HMI tags "2930RS001A01L01"
   "2930RS001A01L01.MSW" : 52809b66-421d-457f-8884-6f7a49d4e247 AT %DB5093.DBX18.0, 500 ms
   "2930RS001A01L01.DefaultText" : TextRef, internal   // Заголовок POPUP окна. При експорте из ECS через скрипт заполняется автоматически, если теги копируются в ручную то требуется в ручную задатать свойство Start Value
   "2930RS001A01L01.BlockInfo" : Array [0..2] of Int AT %DB5093.DBX38.0, 500 ms
   "2930RS001A01L01.StatusWork" : Int AT %DB5093.DBW242, 500 ms
   "2930RS001A01L01.FP_PARAM.DampingTime" : Int AT %DB5093.DBW50, 500 ms
   "2930RS001A01L01.FP_PARAM.Force_Value" : Real AT %DB5093.DBD52, 500 ms
   "2930RS001A01L01.FP_PARAM.Scale_Min" : Real AT %DB5093.DBD56, 500 ms
   "2930RS001A01L01.FP_PARAM.Scale_Max" : Real AT %DB5093.DBD60, 500 ms
   "2930RS001A01L01.FP_PARAM.Gradient" : Real AT %DB5093.DBD64, 500 ms
   "2930RS001A01L01.FP_PARAM.Grad_Pos" : Real AT %DB5093.DBD68, 500 ms
   "2930RS001A01L01.FP_PARAM.Grad_Neg" : Real AT %DB5093.DBD72, 500 ms
   "2930RS001A01L01.FP_PARAM.Grad_X" : Real AT %DB5093.DBD76, 500 ms
   "2930RS001A01L01.FP_PARAM.Gradient_Time_Pre" : Int AT %DB5093.DBW80, 500 ms
   "2930RS001A01L01.FP_PARAM.Gradient_Time_ACC" : Int AT %DB5093.DBW82, 500 ms
   "2930RS001A01L01.FP_PARAM.Alarm_Hyst" : Real AT %DB5093.DBD84, 500 ms
   "2930RS001A01L01.FP_PARAM.AlarmLimit_H3" : Real AT %DB5093.DBD88, 500 ms
   "2930RS001A01L01.FP_PARAM.AlarmLimit_H2" : Real AT %DB5093.DBD92, 500 ms
   "2930RS001A01L01.FP_PARAM.AlarmLimit_H1" : Real AT %DB5093.DBD96, 500 ms
   "2930RS001A01L01.FP_PARAM.AlarmLimit_L1" : Real AT %DB5093.DBD100, 500 ms
   "2930RS001A01L01.FP_PARAM.AlarmLimit_L2" : Real AT %DB5093.DBD104, 500 ms
   "2930RS001A01L01.FP_PARAM.AlarmLimit_L3" : Real AT %DB5093.DBD108, 500 ms
   "2930RS001A01L01.FP_PARAM.AlarmDelay_H3_Pre" : Int AT %DB5093.DBW112, 500 ms
   "2930RS001A01L01.FP_PARAM.AlarmDelay_H3_Acc" : Int AT %DB5093.DBW114, 500 ms
   "2930RS001A01L01.FP_PARAM.AlarmDelay_H2_Pre" : Int AT %DB5093.DBW116, 500 ms
   "2930RS001A01L01.FP_PARAM.AlarmDelay_H2_Acc" : Int AT %DB5093.DBW118, 500 ms
   "2930RS001A01L01.FP_PARAM.AlarmDelay_H1_Pre" : Int AT %DB5093.DBW120, 500 ms
   "2930RS001A01L01.FP_PARAM.AlarmDelay_H1_Acc" : Int AT %DB5093.DBW122, 500 ms
   "2930RS001A01L01.FP_PARAM.AlarmDelay_L1_Pre" : Int AT %DB5093.DBW124, 500 ms
   "2930RS001A01L01.FP_PARAM.AlarmDelay_L1_Acc" : Int AT %DB5093.DBW126, 500 ms
   "2930RS001A01L01.FP_PARAM.AlarmDelay_L2_Pre" : Int AT %DB5093.DBW128, 500 ms
   "2930RS001A01L01.FP_PARAM.AlarmDelay_L2_Acc" : Int AT %DB5093.DBW130, 500 ms
   "2930RS001A01L01.FP_PARAM.AlarmDelay_L3_Pre" : Int AT %DB5093.DBW132, 500 ms
   "2930RS001A01L01.FP_PARAM.AlarmDelay_L3_Acc" : Int AT %DB5093.DBW134, 500 ms
   "2930RS001A01L01.FP_PARAM.OpenLoopDelay_Pre" : Int AT %DB5093.DBW136, 500 ms
   "2930RS001A01L01.FP_PARAM.OpenLoopDelay_Acc" : Int AT %DB5093.DBW138, 500 ms
   "2930RS001A01L01.FP_PARAM.OverRangeDelay_Pre" : Int AT %DB5093.DBW140, 500 ms
   "2930RS001A01L01.FP_PARAM.OverRangeDelay_Acc" : Int AT %DB5093.DBW142, 500 ms
   "2930RS001A01L01.FP_PARAM.AuxLimit_H2_Value" : Real AT %DB5093.DBD144, 500 ms
   "2930RS001A01L01.FP_PARAM.AuxLimit_H1_Value" : Real AT %DB5093.DBD148, 500 ms
   "2930RS001A01L01.FP_PARAM.AuxLimit_L2_Value" : Real AT %DB5093.DBD152, 500 ms
   "2930RS001A01L01.FP_PARAM.AuxLimit_L1_Value" : Real AT %DB5093.DBD156, 500 ms
   "2930RS001A01L01.Unit" : TextRef, internal   // Еденицы измерения При експорте из ECS через скрипт заполняется автоматически, если теги копируются в ручную то требуется задатать свойство Text
   "2930RS001A01L01.Decimals" : TextRef, internal   // Формат отображения При експорте из ECS через скрипт, заполняется автоматически. Если теги копируются в ручную то требуется задатать свойство Text s999999.9
   "2930RS001A01L01.FP_EN.Square" : Bool AT %DB5093.DBX46.0, 500 ms
   "2930RS001A01L01.FP_EN.SquareRoot" : Bool AT %DB5093.DBX46.1, 500 ms
   "2930RS001A01L01.FP_EN.ParentSupress" : Bool AT %DB5093.DBX46.2, 500 ms
   "2930RS001A01L01.FP_EN.ParentSupressUnit" : Bool AT %DB5093.DBX46.3, 500 ms
   "2930RS001A01L01.FP_EN.Force" : Bool AT %DB5093.DBX46.4, 500 ms
   "2930RS001A01L01.FP_EN.Damping" : Bool AT %DB5093.DBX46.5, 500 ms
   "2930RS001A01L01.FP_EN.Gradient_Pos" : Bool AT %DB5093.DBX46.6, 500 ms
   "2930RS001A01L01.FP_EN.Gradient_Neg" : Bool AT %DB5093.DBX46.7, 500 ms
   "2930RS001A01L01.FP_EN.Hysteresis" : Bool AT %DB5093.DBX47.0, 500 ms
   "2930RS001A01L01.FP_EN.Alarm_H3" : Bool AT %DB5093.DBX47.1, 500 ms
   "2930RS001A01L01.FP_EN.Alarm_H2" : Bool AT %DB5093.DBX47.2, 500 ms
   "2930RS001A01L01.FP_EN.Alarm_H1" : Bool AT %DB5093.DBX47.3, 500 ms
   "2930RS001A01L01.FP_EN.Alarm_L1" : Bool AT %DB5093.DBX47.4, 500 ms
   "2930RS001A01L01.FP_EN.Alarm_L2" : Bool AT %DB5093.DBX47.5, 500 ms
   "2930RS001A01L01.FP_EN.Alarm_L3" : Bool AT %DB5093.DBX47.6, 500 ms
   "2930RS001A01L01.FP_EN.AlarmDelay_H3" : Bool AT %DB5093.DBX47.7, 500 ms
   "2930RS001A01L01.FP_EN.AlarmDelay_H2" : Bool AT %DB5093.DBX48.0, 500 ms
   "2930RS001A01L01.FP_EN.AlarmDelay_H1" : Bool AT %DB5093.DBX48.1, 500 ms
   "2930RS001A01L01.FP_EN.AlarmDelay_L1" : Bool AT %DB5093.DBX48.2, 500 ms
   "2930RS001A01L01.FP_EN.AlarmDelay_L2" : Bool AT %DB5093.DBX48.3, 500 ms
   "2930RS001A01L01.FP_EN.AlarmDelay_L3" : Bool AT %DB5093.DBX48.4, 500 ms
   "2930RS001A01L01.FP_EN.ROC_Warn" : Bool AT %DB5093.DBX48.5, 500 ms
   "2930RS001A01L01.FP_EN.U_Range_Warn" : Bool AT %DB5093.DBX48.6, 500 ms
   "2930RS001A01L01.FP_EN.O_Range_Warn" : Bool AT %DB5093.DBX48.7, 500 ms
   "2930RS001A01L01.trend_tag_name" : TextRef, internal   // Еденицы измерения При експорте из ECS через скрипт - заполняется автоматически, если теги копируются в ручную то требуется задатать свойство Text - имя тега для тренда
   "2930RS001A01L01.DQ.AL_H3" : Bool AT %DB5093.DBX16.0, 500 ms
   "2930RS001A01L01.DQ.AL_H2" : Bool AT %DB5093.DBX16.1, 500 ms
   "2930RS001A01L01.DQ.AL_H1" : Bool AT %DB5093.DBX16.2, 500 ms
   "2930RS001A01L01.DQ.AL_L1" : Bool AT %DB5093.DBX16.3, 500 ms
   "2930RS001A01L01.DQ.AL_L2" : Bool AT %DB5093.DBX16.4, 500 ms
   "2930RS001A01L01.DQ.AL_L3" : Bool AT %DB5093.DBX16.5, 500 ms
   "2930RS001A01L01.DQ.SIG_OK" : Bool AT %DB5093.DBX16.6, 500 ms
   "2930RS001A01L01.DQ.LIM_H2" : Bool AT %DB5093.DBX16.7, 500 ms
   "2930RS001A01L01.DQ.LIM_H1" : Bool AT %DB5093.DBX17.0, 500 ms
   "2930RS001A01L01.DQ.LIM_L1" : Bool AT %DB5093.DBX17.1, 500 ms
   "2930RS001A01L01.DQ.LIM_L2" : Bool AT %DB5093.DBX17.2, 500 ms
   "2930RS001A01L01.DQ.GR_P" : Bool AT %DB5093.DBX17.3, 500 ms
   "2930RS001A01L01.DQ.GR_N" : Bool AT %DB5093.DBX17.4, 500 ms
   "2930RS001A01L01.I.IN" : Real AT %DB5093.DBD2, 500 ms
   "2930RS001A01L01.I.SIG_TYPE" : Int AT %DB5093.DBW0, 500 ms
   "2930RS001A01L01.I.FI_BUS" : Byte AT %DB5093.DBB6, 500 ms
   "2930RS001A01L01.DI.U_RANGE" : Bool AT %DB5093.DBX7.0, 500 ms
   "2930RS001A01L01.DI.O_RANGE" : Bool AT %DB5093.DBX7.1, 500 ms
   "2930RS001A01L01.DI.SIG_FAULT" : Bool AT %DB5093.DBX7.2, 500 ms
   "2930RS001A01L01.DI.EnConfig" : Bool AT %DB5093.DBX7.3, 500 ms
   "2930RS001A01L01.DI.AEN" : Bool AT %DB5093.DBX7.4, 500 ms
   "2930RS001A01L01.DI.AL_SUPR" : Bool AT %DB5093.DBX7.5, 500 ms
   "2930RS001A01L01.Q.PV_NORM" : Real AT %DB5093.DBD8, 500 ms
   "2930RS001A01L01.Q.PV_SCAL" : Real AT %DB5093.DBD12, 500 ms
   "2930RS001A01L01.ParentInfo" : TextRef, internal   // Имя родителя для попап окна, вкладка инфо. При експорте из ECS через скрипт заполняется автоматически, если теги копируются в ручную то требуется в ручную задатать свойство Start Value

HMI tags "2930RS001A01L02"
   "2930RS001A01L02.MSW" : 52809b66-421d-457f-8884-6f7a49d4e247 AT %DB5094.DBX18.0, 500 ms
   "2930RS001A01L02.DefaultText" : TextRef, internal   // Заголовок POPUP окна. При експорте из ECS через скрипт заполняется автоматически, если теги копируются в ручную то требуется в ручную задатать свойство Start Value
   "2930RS001A01L02.BlockInfo" : Array [0..2] of Int AT %DB5094.DBX38.0, 500 ms
   "2930RS001A01L02.StatusWork" : Int AT %DB5094.DBW242, 500 ms
   "2930RS001A01L02.FP_PARAM.DampingTime" : Int AT %DB5094.DBW50, 500 ms
   "2930RS001A01L02.FP_PARAM.Force_Value" : Real AT %DB5094.DBD52, 500 ms
   "2930RS001A01L02.FP_PARAM.Scale_Min" : Real AT %DB5094.DBD56, 500 ms
   "2930RS001A01L02.FP_PARAM.Scale_Max" : Real AT %DB5094.DBD60, 500 ms
   "2930RS001A01L02.FP_PARAM.Gradient" : Real AT %DB5094.DBD64, 500 ms
   "2930RS001A01L02.FP_PARAM.Grad_Pos" : Real AT %DB5094.DBD68, 500 ms
   "2930RS001A01L02.FP_PARAM.Grad_Neg" : Real AT %DB5094.DBD72, 500 ms
   "2930RS001A01L02.FP_PARAM.Grad_X" : Real AT %DB5094.DBD76, 500 ms
   "2930RS001A01L02.FP_PARAM.Gradient_Time_Pre" : Int AT %DB5094.DBW80, 500 ms
   "2930RS001A01L02.FP_PARAM.Gradient_Time_ACC" : Int AT %DB5094.DBW82, 500 ms
   "2930RS001A01L02.FP_PARAM.Alarm_Hyst" : Real AT %DB5094.DBD84, 500 ms
   "2930RS001A01L02.FP_PARAM.AlarmLimit_H3" : Real AT %DB5094.DBD88, 500 ms
   "2930RS001A01L02.FP_PARAM.AlarmLimit_H2" : Real AT %DB5094.DBD92, 500 ms
   "2930RS001A01L02.FP_PARAM.AlarmLimit_H1" : Real AT %DB5094.DBD96, 500 ms
   "2930RS001A01L02.FP_PARAM.AlarmLimit_L1" : Real AT %DB5094.DBD100, 500 ms
   "2930RS001A01L02.FP_PARAM.AlarmLimit_L2" : Real AT %DB5094.DBD104, 500 ms
   "2930RS001A01L02.FP_PARAM.AlarmLimit_L3" : Real AT %DB5094.DBD108, 500 ms
   "2930RS001A01L02.FP_PARAM.AlarmDelay_H3_Pre" : Int AT %DB5094.DBW112, 500 ms
   "2930RS001A01L02.FP_PARAM.AlarmDelay_H3_Acc" : Int AT %DB5094.DBW114, 500 ms
   "2930RS001A01L02.FP_PARAM.AlarmDelay_H2_Pre" : Int AT %DB5094.DBW116, 500 ms
   "2930RS001A01L02.FP_PARAM.AlarmDelay_H2_Acc" : Int AT %DB5094.DBW118, 500 ms
   "2930RS001A01L02.FP_PARAM.AlarmDelay_H1_Pre" : Int AT %DB5094.DBW120, 500 ms
   "2930RS001A01L02.FP_PARAM.AlarmDelay_H1_Acc" : Int AT %DB5094.DBW122, 500 ms
   "2930RS001A01L02.FP_PARAM.AlarmDelay_L1_Pre" : Int AT %DB5094.DBW124, 500 ms
   "2930RS001A01L02.FP_PARAM.AlarmDelay_L1_Acc" : Int AT %DB5094.DBW126, 500 ms
   "2930RS001A01L02.FP_PARAM.AlarmDelay_L2_Pre" : Int AT %DB5094.DBW128, 500 ms
   "2930RS001A01L02.FP_PARAM.AlarmDelay_L2_Acc" : Int AT %DB5094.DBW130, 500 ms
   "2930RS001A01L02.FP_PARAM.AlarmDelay_L3_Pre" : Int AT %DB5094.DBW132, 500 ms
   "2930RS001A01L02.FP_PARAM.AlarmDelay_L3_Acc" : Int AT %DB5094.DBW134, 500 ms
   "2930RS001A01L02.FP_PARAM.OpenLoopDelay_Pre" : Int AT %DB5094.DBW136, 500 ms
   "2930RS001A01L02.FP_PARAM.OpenLoopDelay_Acc" : Int AT %DB5094.DBW138, 500 ms
   "2930RS001A01L02.FP_PARAM.OverRangeDelay_Pre" : Int AT %DB5094.DBW140, 500 ms
   "2930RS001A01L02.FP_PARAM.OverRangeDelay_Acc" : Int AT %DB5094.DBW142, 500 ms
   "2930RS001A01L02.FP_PARAM.AuxLimit_H2_Value" : Real AT %DB5094.DBD144, 500 ms
   "2930RS001A01L02.FP_PARAM.AuxLimit_H1_Value" : Real AT %DB5094.DBD148, 500 ms
   "2930RS001A01L02.FP_PARAM.AuxLimit_L2_Value" : Real AT %DB5094.DBD152, 500 ms
   "2930RS001A01L02.FP_PARAM.AuxLimit_L1_Value" : Real AT %DB5094.DBD156, 500 ms
   "2930RS001A01L02.Unit" : TextRef, internal   // Еденицы измерения При експорте из ECS через скрипт заполняется автоматически, если теги копируются в ручную то требуется задатать свойство Text
   "2930RS001A01L02.Decimals" : TextRef, internal   // Формат отображения При експорте из ECS через скрипт, заполняется автоматически. Если теги копируются в ручную то требуется задатать свойство Text s999999.9
   "2930RS001A01L02.FP_EN.Square" : Bool AT %DB5094.DBX46.0, 500 ms
   "2930RS001A01L02.FP_EN.SquareRoot" : Bool AT %DB5094.DBX46.1, 500 ms
   "2930RS001A01L02.FP_EN.ParentSupress" : Bool AT %DB5094.DBX46.2, 500 ms
   "2930RS001A01L02.FP_EN.ParentSupressUnit" : Bool AT %DB5094.DBX46.3, 500 ms
   "2930RS001A01L02.FP_EN.Force" : Bool AT %DB5094.DBX46.4, 500 ms
   "2930RS001A01L02.FP_EN.Damping" : Bool AT %DB5094.DBX46.5, 500 ms
   "2930RS001A01L02.FP_EN.Gradient_Pos" : Bool AT %DB5094.DBX46.6, 500 ms
   "2930RS001A01L02.FP_EN.Gradient_Neg" : Bool AT %DB5094.DBX46.7, 500 ms
   "2930RS001A01L02.FP_EN.Hysteresis" : Bool AT %DB5094.DBX47.0, 500 ms
   "2930RS001A01L02.FP_EN.Alarm_H3" : Bool AT %DB5094.DBX47.1, 500 ms
   "2930RS001A01L02.FP_EN.Alarm_H2" : Bool AT %DB5094.DBX47.2, 500 ms
   "2930RS001A01L02.FP_EN.Alarm_H1" : Bool AT %DB5094.DBX47.3, 500 ms
   "2930RS001A01L02.FP_EN.Alarm_L1" : Bool AT %DB5094.DBX47.4, 500 ms
   "2930RS001A01L02.FP_EN.Alarm_L2" : Bool AT %DB5094.DBX47.5, 500 ms
   "2930RS001A01L02.FP_EN.Alarm_L3" : Bool AT %DB5094.DBX47.6, 500 ms
   "2930RS001A01L02.FP_EN.AlarmDelay_H3" : Bool AT %DB5094.DBX47.7, 500 ms
   "2930RS001A01L02.FP_EN.AlarmDelay_H2" : Bool AT %DB5094.DBX48.0, 500 ms
   "2930RS001A01L02.FP_EN.AlarmDelay_H1" : Bool AT %DB5094.DBX48.1, 500 ms
   "2930RS001A01L02.FP_EN.AlarmDelay_L1" : Bool AT %DB5094.DBX48.2, 500 ms
   "2930RS001A01L02.FP_EN.AlarmDelay_L2" : Bool AT %DB5094.DBX48.3, 500 ms
   "2930RS001A01L02.FP_EN.AlarmDelay_L3" : Bool AT %DB5094.DBX48.4, 500 ms
   "2930RS001A01L02.FP_EN.ROC_Warn" : Bool AT %DB5094.DBX48.5, 500 ms
   "2930RS001A01L02.FP_EN.U_Range_Warn" : Bool AT %DB5094.DBX48.6, 500 ms
   "2930RS001A01L02.FP_EN.O_Range_Warn" : Bool AT %DB5094.DBX48.7, 500 ms
   "2930RS001A01L02.trend_tag_name" : TextRef, internal   // Еденицы измерения При експорте из ECS через скрипт - заполняется автоматически, если теги копируются в ручную то требуется задатать свойство Text - имя тега для тренда
   "2930RS001A01L02.DQ.AL_H3" : Bool AT %DB5094.DBX16.0, 500 ms
   "2930RS001A01L02.DQ.AL_H2" : Bool AT %DB5094.DBX16.1, 500 ms
   "2930RS001A01L02.DQ.AL_H1" : Bool AT %DB5094.DBX16.2, 500 ms
   "2930RS001A01L02.DQ.AL_L1" : Bool AT %DB5094.DBX16.3, 500 ms
   "2930RS001A01L02.DQ.AL_L2" : Bool AT %DB5094.DBX16.4, 500 ms
   "2930RS001A01L02.DQ.AL_L3" : Bool AT %DB5094.DBX16.5, 500 ms
   "2930RS001A01L02.DQ.SIG_OK" : Bool AT %DB5094.DBX16.6, 500 ms
   "2930RS001A01L02.DQ.LIM_H2" : Bool AT %DB5094.DBX16.7, 500 ms
   "2930RS001A01L02.DQ.LIM_H1" : Bool AT %DB5094.DBX17.0, 500 ms
   "2930RS001A01L02.DQ.LIM_L1" : Bool AT %DB5094.DBX17.1, 500 ms
   "2930RS001A01L02.DQ.LIM_L2" : Bool AT %DB5094.DBX17.2, 500 ms
   "2930RS001A01L02.DQ.GR_P" : Bool AT %DB5094.DBX17.3, 500 ms
   "2930RS001A01L02.DQ.GR_N" : Bool AT %DB5094.DBX17.4, 500 ms
   "2930RS001A01L02.I.IN" : Real AT %DB5094.DBD2, 500 ms
   "2930RS001A01L02.I.SIG_TYPE" : Int AT %DB5094.DBW0, 500 ms
   "2930RS001A01L02.I.FI_BUS" : Byte AT %DB5094.DBB6, 500 ms
   "2930RS001A01L02.DI.U_RANGE" : Bool AT %DB5094.DBX7.0, 500 ms
   "2930RS001A01L02.DI.O_RANGE" : Bool AT %DB5094.DBX7.1, 500 ms
   "2930RS001A01L02.DI.SIG_FAULT" : Bool AT %DB5094.DBX7.2, 500 ms
   "2930RS001A01L02.DI.EnConfig" : Bool AT %DB5094.DBX7.3, 500 ms
   "2930RS001A01L02.DI.AEN" : Bool AT %DB5094.DBX7.4, 500 ms
   "2930RS001A01L02.DI.AL_SUPR" : Bool AT %DB5094.DBX7.5, 500 ms
   "2930RS001A01L02.Q.PV_NORM" : Real AT %DB5094.DBD8, 500 ms
   "2930RS001A01L02.Q.PV_SCAL" : Real AT %DB5094.DBD12, 500 ms
   "2930RS001A01L02.ParentInfo" : TextRef, internal   // Имя родителя для попап окна, вкладка инфо. При експорте из ECS через скрипт заполняется автоматически, если теги копируются в ручную то требуется в ручную задатать свойство Start Value

HMI tags "2930RS001A01P01"
   "2930RS001A01P01.MSW" : 52809b66-421d-457f-8884-6f7a49d4e247 AT %DB5095.DBX18.0, 500 ms
   "2930RS001A01P01.DefaultText" : TextRef, internal   // Заголовок POPUP окна. При експорте из ECS через скрипт заполняется автоматически, если теги копируются в ручную то требуется в ручную задатать свойство Start Value
   "2930RS001A01P01.BlockInfo" : Array [0..2] of Int AT %DB5095.DBX38.0, 500 ms
   "2930RS001A01P01.StatusWork" : Int AT %DB5095.DBW242, 500 ms
   "2930RS001A01P01.FP_PARAM.DampingTime" : Int AT %DB5095.DBW50, 500 ms
   "2930RS001A01P01.FP_PARAM.Force_Value" : Real AT %DB5095.DBD52, 500 ms
   "2930RS001A01P01.FP_PARAM.Scale_Min" : Real AT %DB5095.DBD56, 500 ms
   "2930RS001A01P01.FP_PARAM.Scale_Max" : Real AT %DB5095.DBD60, 500 ms
   "2930RS001A01P01.FP_PARAM.Gradient" : Real AT %DB5095.DBD64, 500 ms
   "2930RS001A01P01.FP_PARAM.Grad_Pos" : Real AT %DB5095.DBD68, 500 ms
   "2930RS001A01P01.FP_PARAM.Grad_Neg" : Real AT %DB5095.DBD72, 500 ms
   "2930RS001A01P01.FP_PARAM.Grad_X" : Real AT %DB5095.DBD76, 500 ms
   "2930RS001A01P01.FP_PARAM.Gradient_Time_Pre" : Int AT %DB5095.DBW80, 500 ms
   "2930RS001A01P01.FP_PARAM.Gradient_Time_ACC" : Int AT %DB5095.DBW82, 500 ms
   "2930RS001A01P01.FP_PARAM.Alarm_Hyst" : Real AT %DB5095.DBD84, 500 ms
   "2930RS001A01P01.FP_PARAM.AlarmLimit_H3" : Real AT %DB5095.DBD88, 500 ms
   "2930RS001A01P01.FP_PARAM.AlarmLimit_H2" : Real AT %DB5095.DBD92, 500 ms
   "2930RS001A01P01.FP_PARAM.AlarmLimit_H1" : Real AT %DB5095.DBD96, 500 ms
   "2930RS001A01P01.FP_PARAM.AlarmLimit_L1" : Real AT %DB5095.DBD100, 500 ms
   "2930RS001A01P01.FP_PARAM.AlarmLimit_L2" : Real AT %DB5095.DBD104, 500 ms
   "2930RS001A01P01.FP_PARAM.AlarmLimit_L3" : Real AT %DB5095.DBD108, 500 ms
   "2930RS001A01P01.FP_PARAM.AlarmDelay_H3_Pre" : Int AT %DB5095.DBW112, 500 ms
   "2930RS001A01P01.FP_PARAM.AlarmDelay_H3_Acc" : Int AT %DB5095.DBW114, 500 ms
   "2930RS001A01P01.FP_PARAM.AlarmDelay_H2_Pre" : Int AT %DB5095.DBW116, 500 ms
   "2930RS001A01P01.FP_PARAM.AlarmDelay_H2_Acc" : Int AT %DB5095.DBW118, 500 ms
   "2930RS001A01P01.FP_PARAM.AlarmDelay_H1_Pre" : Int AT %DB5095.DBW120, 500 ms
   "2930RS001A01P01.FP_PARAM.AlarmDelay_H1_Acc" : Int AT %DB5095.DBW122, 500 ms
   "2930RS001A01P01.FP_PARAM.AlarmDelay_L1_Pre" : Int AT %DB5095.DBW124, 500 ms
   "2930RS001A01P01.FP_PARAM.AlarmDelay_L1_Acc" : Int AT %DB5095.DBW126, 500 ms
   "2930RS001A01P01.FP_PARAM.AlarmDelay_L2_Pre" : Int AT %DB5095.DBW128, 500 ms
   "2930RS001A01P01.FP_PARAM.AlarmDelay_L2_Acc" : Int AT %DB5095.DBW130, 500 ms
   "2930RS001A01P01.FP_PARAM.AlarmDelay_L3_Pre" : Int AT %DB5095.DBW132, 500 ms
   "2930RS001A01P01.FP_PARAM.AlarmDelay_L3_Acc" : Int AT %DB5095.DBW134, 500 ms
   "2930RS001A01P01.FP_PARAM.OpenLoopDelay_Pre" : Int AT %DB5095.DBW136, 500 ms
   "2930RS001A01P01.FP_PARAM.OpenLoopDelay_Acc" : Int AT %DB5095.DBW138, 500 ms
   "2930RS001A01P01.FP_PARAM.OverRangeDelay_Pre" : Int AT %DB5095.DBW140, 500 ms
   "2930RS001A01P01.FP_PARAM.OverRangeDelay_Acc" : Int AT %DB5095.DBW142, 500 ms
   "2930RS001A01P01.FP_PARAM.AuxLimit_H2_Value" : Real AT %DB5095.DBD144, 500 ms
   "2930RS001A01P01.FP_PARAM.AuxLimit_H1_Value" : Real AT %DB5095.DBD148, 500 ms
   "2930RS001A01P01.FP_PARAM.AuxLimit_L2_Value" : Real AT %DB5095.DBD152, 500 ms
   "2930RS001A01P01.FP_PARAM.AuxLimit_L1_Value" : Real AT %DB5095.DBD156, 500 ms
   "2930RS001A01P01.Unit" : TextRef, internal   // Еденицы измерения При експорте из ECS через скрипт заполняется автоматически, если теги копируются в ручную то требуется задатать свойство Text
   "2930RS001A01P01.Decimals" : TextRef, internal   // Формат отображения При експорте из ECS через скрипт, заполняется автоматически. Если теги копируются в ручную то требуется задатать свойство Text s999999.9
   "2930RS001A01P01.FP_EN.Square" : Bool AT %DB5095.DBX46.0, 500 ms
   "2930RS001A01P01.FP_EN.SquareRoot" : Bool AT %DB5095.DBX46.1, 500 ms
   "2930RS001A01P01.FP_EN.ParentSupress" : Bool AT %DB5095.DBX46.2, 500 ms
   "2930RS001A01P01.FP_EN.ParentSupressUnit" : Bool AT %DB5095.DBX46.3, 500 ms
   "2930RS001A01P01.FP_EN.Force" : Bool AT %DB5095.DBX46.4, 500 ms
   "2930RS001A01P01.FP_EN.Damping" : Bool AT %DB5095.DBX46.5, 500 ms
   "2930RS001A01P01.FP_EN.Gradient_Pos" : Bool AT %DB5095.DBX46.6, 500 ms
   "2930RS001A01P01.FP_EN.Gradient_Neg" : Bool AT %DB5095.DBX46.7, 500 ms
   "2930RS001A01P01.FP_EN.Hysteresis" : Bool AT %DB5095.DBX47.0, 500 ms
   "2930RS001A01P01.FP_EN.Alarm_H3" : Bool AT %DB5095.DBX47.1, 500 ms
   "2930RS001A01P01.FP_EN.Alarm_H2" : Bool AT %DB5095.DBX47.2, 500 ms
   "2930RS001A01P01.FP_EN.Alarm_H1" : Bool AT %DB5095.DBX47.3, 500 ms
   "2930RS001A01P01.FP_EN.Alarm_L1" : Bool AT %DB5095.DBX47.4, 500 ms
   "2930RS001A01P01.FP_EN.Alarm_L2" : Bool AT %DB5095.DBX47.5, 500 ms
   "2930RS001A01P01.FP_EN.Alarm_L3" : Bool AT %DB5095.DBX47.6, 500 ms
   "2930RS001A01P01.FP_EN.AlarmDelay_H3" : Bool AT %DB5095.DBX47.7, 500 ms
   "2930RS001A01P01.FP_EN.AlarmDelay_H2" : Bool AT %DB5095.DBX48.0, 500 ms
   "2930RS001A01P01.FP_EN.AlarmDelay_H1" : Bool AT %DB5095.DBX48.1, 500 ms
   "2930RS001A01P01.FP_EN.AlarmDelay_L1" : Bool AT %DB5095.DBX48.2, 500 ms
   "2930RS001A01P01.FP_EN.AlarmDelay_L2" : Bool AT %DB5095.DBX48.3, 500 ms
   "2930RS001A01P01.FP_EN.AlarmDelay_L3" : Bool AT %DB5095.DBX48.4, 500 ms
   "2930RS001A01P01.FP_EN.ROC_Warn" : Bool AT %DB5095.DBX48.5, 500 ms
   "2930RS001A01P01.FP_EN.U_Range_Warn" : Bool AT %DB5095.DBX48.6, 500 ms
   "2930RS001A01P01.FP_EN.O_Range_Warn" : Bool AT %DB5095.DBX48.7, 500 ms
   "2930RS001A01P01.trend_tag_name" : TextRef, internal   // Еденицы измерения При експорте из ECS через скрипт - заполняется автоматически, если теги копируются в ручную то требуется задатать свойство Text - имя тега для тренда
   "2930RS001A01P01.DQ.AL_H3" : Bool AT %DB5095.DBX16.0, 500 ms
   "2930RS001A01P01.DQ.AL_H2" : Bool AT %DB5095.DBX16.1, 500 ms
   "2930RS001A01P01.DQ.AL_H1" : Bool AT %DB5095.DBX16.2, 500 ms
   "2930RS001A01P01.DQ.AL_L1" : Bool AT %DB5095.DBX16.3, 500 ms
   "2930RS001A01P01.DQ.AL_L2" : Bool AT %DB5095.DBX16.4, 500 ms
   "2930RS001A01P01.DQ.AL_L3" : Bool AT %DB5095.DBX16.5, 500 ms
   "2930RS001A01P01.DQ.SIG_OK" : Bool AT %DB5095.DBX16.6, 500 ms
   "2930RS001A01P01.DQ.LIM_H2" : Bool AT %DB5095.DBX16.7, 500 ms
   "2930RS001A01P01.DQ.LIM_H1" : Bool AT %DB5095.DBX17.0, 500 ms
   "2930RS001A01P01.DQ.LIM_L1" : Bool AT %DB5095.DBX17.1, 500 ms
   "2930RS001A01P01.DQ.LIM_L2" : Bool AT %DB5095.DBX17.2, 500 ms
   "2930RS001A01P01.DQ.GR_P" : Bool AT %DB5095.DBX17.3, 500 ms
   "2930RS001A01P01.DQ.GR_N" : Bool AT %DB5095.DBX17.4, 500 ms
   "2930RS001A01P01.I.IN" : Real AT %DB5095.DBD2, 500 ms
   "2930RS001A01P01.I.SIG_TYPE" : Int AT %DB5095.DBW0, 500 ms
   "2930RS001A01P01.I.FI_BUS" : Byte AT %DB5095.DBB6, 500 ms
   "2930RS001A01P01.DI.U_RANGE" : Bool AT %DB5095.DBX7.0, 500 ms
   "2930RS001A01P01.DI.O_RANGE" : Bool AT %DB5095.DBX7.1, 500 ms
   "2930RS001A01P01.DI.SIG_FAULT" : Bool AT %DB5095.DBX7.2, 500 ms
   "2930RS001A01P01.DI.EnConfig" : Bool AT %DB5095.DBX7.3, 500 ms
   "2930RS001A01P01.DI.AEN" : Bool AT %DB5095.DBX7.4, 500 ms
   "2930RS001A01P01.DI.AL_SUPR" : Bool AT %DB5095.DBX7.5, 500 ms
   "2930RS001A01P01.Q.PV_NORM" : Real AT %DB5095.DBD8, 500 ms
   "2930RS001A01P01.Q.PV_SCAL" : Real AT %DB5095.DBD12, 500 ms
   "2930RS001A01P01.ParentInfo" : TextRef, internal   // Имя родителя для попап окна, вкладка инфо. При експорте из ECS через скрипт заполняется автоматически, если теги копируются в ручную то требуется в ручную задатать свойство Start Value

HMI tags "2930RS001A01T01"
   "2930RS001A01T01.MSW" : 52809b66-421d-457f-8884-6f7a49d4e247 AT %DB5096.DBX18.0, 500 ms
   "2930RS001A01T01.DefaultText" : TextRef, internal   // Заголовок POPUP окна. При експорте из ECS через скрипт заполняется автоматически, если теги копируются в ручную то требуется в ручную задатать свойство Start Value
   "2930RS001A01T01.BlockInfo" : Array [0..2] of Int AT %DB5096.DBX38.0, 500 ms
   "2930RS001A01T01.StatusWork" : Int AT %DB5096.DBW242, 500 ms
   "2930RS001A01T01.FP_PARAM.DampingTime" : Int AT %DB5096.DBW50, 500 ms
   "2930RS001A01T01.FP_PARAM.Force_Value" : Real AT %DB5096.DBD52, 500 ms
   "2930RS001A01T01.FP_PARAM.Scale_Min" : Real AT %DB5096.DBD56, 500 ms
   "2930RS001A01T01.FP_PARAM.Scale_Max" : Real AT %DB5096.DBD60, 500 ms
   "2930RS001A01T01.FP_PARAM.Gradient" : Real AT %DB5096.DBD64, 500 ms
   "2930RS001A01T01.FP_PARAM.Grad_Pos" : Real AT %DB5096.DBD68, 500 ms
   "2930RS001A01T01.FP_PARAM.Grad_Neg" : Real AT %DB5096.DBD72, 500 ms
   "2930RS001A01T01.FP_PARAM.Grad_X" : Real AT %DB5096.DBD76, 500 ms
   "2930RS001A01T01.FP_PARAM.Gradient_Time_Pre" : Int AT %DB5096.DBW80, 500 ms
   "2930RS001A01T01.FP_PARAM.Gradient_Time_ACC" : Int AT %DB5096.DBW82, 500 ms
   "2930RS001A01T01.FP_PARAM.Alarm_Hyst" : Real AT %DB5096.DBD84, 500 ms
   "2930RS001A01T01.FP_PARAM.AlarmLimit_H3" : Real AT %DB5096.DBD88, 500 ms
   "2930RS001A01T01.FP_PARAM.AlarmLimit_H2" : Real AT %DB5096.DBD92, 500 ms
   "2930RS001A01T01.FP_PARAM.AlarmLimit_H1" : Real AT %DB5096.DBD96, 500 ms
   "2930RS001A01T01.FP_PARAM.AlarmLimit_L1" : Real AT %DB5096.DBD100, 500 ms
   "2930RS001A01T01.FP_PARAM.AlarmLimit_L2" : Real AT %DB5096.DBD104, 500 ms
   "2930RS001A01T01.FP_PARAM.AlarmLimit_L3" : Real AT %DB5096.DBD108, 500 ms
   "2930RS001A01T01.FP_PARAM.AlarmDelay_H3_Pre" : Int AT %DB5096.DBW112, 500 ms
   "2930RS001A01T01.FP_PARAM.AlarmDelay_H3_Acc" : Int AT %DB5096.DBW114, 500 ms
   "2930RS001A01T01.FP_PARAM.AlarmDelay_H2_Pre" : Int AT %DB5096.DBW116, 500 ms
   "2930RS001A01T01.FP_PARAM.AlarmDelay_H2_Acc" : Int AT %DB5096.DBW118, 500 ms
   "2930RS001A01T01.FP_PARAM.AlarmDelay_H1_Pre" : Int AT %DB5096.DBW120, 500 ms
   "2930RS001A01T01.FP_PARAM.AlarmDelay_H1_Acc" : Int AT %DB5096.DBW122, 500 ms
   "2930RS001A01T01.FP_PARAM.AlarmDelay_L1_Pre" : Int AT %DB5096.DBW124, 500 ms
   "2930RS001A01T01.FP_PARAM.AlarmDelay_L1_Acc" : Int AT %DB5096.DBW126, 500 ms
   "2930RS001A01T01.FP_PARAM.AlarmDelay_L2_Pre" : Int AT %DB5096.DBW128, 500 ms
   "2930RS001A01T01.FP_PARAM.AlarmDelay_L2_Acc" : Int AT %DB5096.DBW130, 500 ms
   "2930RS001A01T01.FP_PARAM.AlarmDelay_L3_Pre" : Int AT %DB5096.DBW132, 500 ms
   "2930RS001A01T01.FP_PARAM.AlarmDelay_L3_Acc" : Int AT %DB5096.DBW134, 500 ms
   "2930RS001A01T01.FP_PARAM.OpenLoopDelay_Pre" : Int AT %DB5096.DBW136, 500 ms
   "2930RS001A01T01.FP_PARAM.OpenLoopDelay_Acc" : Int AT %DB5096.DBW138, 500 ms
   "2930RS001A01T01.FP_PARAM.OverRangeDelay_Pre" : Int AT %DB5096.DBW140, 500 ms
   "2930RS001A01T01.FP_PARAM.OverRangeDelay_Acc" : Int AT %DB5096.DBW142, 500 ms
   "2930RS001A01T01.FP_PARAM.AuxLimit_H2_Value" : Real AT %DB5096.DBD144, 500 ms
   "2930RS001A01T01.FP_PARAM.AuxLimit_H1_Value" : Real AT %DB5096.DBD148, 500 ms
   "2930RS001A01T01.FP_PARAM.AuxLimit_L2_Value" : Real AT %DB5096.DBD152, 500 ms
   "2930RS001A01T01.FP_PARAM.AuxLimit_L1_Value" : Real AT %DB5096.DBD156, 500 ms
   "2930RS001A01T01.Unit" : TextRef, internal   // Еденицы измерения При експорте из ECS через скрипт заполняется автоматически, если теги копируются в ручную то требуется задатать свойство Text
   "2930RS001A01T01.Decimals" : TextRef, internal   // Формат отображения При експорте из ECS через скрипт, заполняется автоматически. Если теги копируются в ручную то требуется задатать свойство Text s999999.9
   "2930RS001A01T01.FP_EN.Square" : Bool AT %DB5096.DBX46.0, 500 ms
   "2930RS001A01T01.FP_EN.SquareRoot" : Bool AT %DB5096.DBX46.1, 500 ms
   "2930RS001A01T01.FP_EN.ParentSupress" : Bool AT %DB5096.DBX46.2, 500 ms
   "2930RS001A01T01.FP_EN.ParentSupressUnit" : Bool AT %DB5096.DBX46.3, 500 ms
   "2930RS001A01T01.FP_EN.Force" : Bool AT %DB5096.DBX46.4, 500 ms
   "2930RS001A01T01.FP_EN.Damping" : Bool AT %DB5096.DBX46.5, 500 ms
   "2930RS001A01T01.FP_EN.Gradient_Pos" : Bool AT %DB5096.DBX46.6, 500 ms
   "2930RS001A01T01.FP_EN.Gradient_Neg" : Bool AT %DB5096.DBX46.7, 500 ms
   "2930RS001A01T01.FP_EN.Hysteresis" : Bool AT %DB5096.DBX47.0, 500 ms
   "2930RS001A01T01.FP_EN.Alarm_H3" : Bool AT %DB5096.DBX47.1, 500 ms
   "2930RS001A01T01.FP_EN.Alarm_H2" : Bool AT %DB5096.DBX47.2, 500 ms
   "2930RS001A01T01.FP_EN.Alarm_H1" : Bool AT %DB5096.DBX47.3, 500 ms
   "2930RS001A01T01.FP_EN.Alarm_L1" : Bool AT %DB5096.DBX47.4, 500 ms
   "2930RS001A01T01.FP_EN.Alarm_L2" : Bool AT %DB5096.DBX47.5, 500 ms
   "2930RS001A01T01.FP_EN.Alarm_L3" : Bool AT %DB5096.DBX47.6, 500 ms
   "2930RS001A01T01.FP_EN.AlarmDelay_H3" : Bool AT %DB5096.DBX47.7, 500 ms
   "2930RS001A01T01.FP_EN.AlarmDelay_H2" : Bool AT %DB5096.DBX48.0, 500 ms
   "2930RS001A01T01.FP_EN.AlarmDelay_H1" : Bool AT %DB5096.DBX48.1, 500 ms
   "2930RS001A01T01.FP_EN.AlarmDelay_L1" : Bool AT %DB5096.DBX48.2, 500 ms
   "2930RS001A01T01.FP_EN.AlarmDelay_L2" : Bool AT %DB5096.DBX48.3, 500 ms
   "2930RS001A01T01.FP_EN.AlarmDelay_L3" : Bool AT %DB5096.DBX48.4, 500 ms
   "2930RS001A01T01.FP_EN.ROC_Warn" : Bool AT %DB5096.DBX48.5, 500 ms
   "2930RS001A01T01.FP_EN.U_Range_Warn" : Bool AT %DB5096.DBX48.6, 500 ms
   "2930RS001A01T01.FP_EN.O_Range_Warn" : Bool AT %DB5096.DBX48.7, 500 ms
   "2930RS001A01T01.trend_tag_name" : TextRef, internal   // Еденицы измерения При експорте из ECS через скрипт - заполняется автоматически, если теги копируются в ручную то требуется задатать свойство Text - имя тега для тренда
   "2930RS001A01T01.DQ.AL_H3" : Bool AT %DB5096.DBX16.0, 500 ms
   "2930RS001A01T01.DQ.AL_H2" : Bool AT %DB5096.DBX16.1, 500 ms
   "2930RS001A01T01.DQ.AL_H1" : Bool AT %DB5096.DBX16.2, 500 ms
   "2930RS001A01T01.DQ.AL_L1" : Bool AT %DB5096.DBX16.3, 500 ms
   "2930RS001A01T01.DQ.AL_L2" : Bool AT %DB5096.DBX16.4, 500 ms
   "2930RS001A01T01.DQ.AL_L3" : Bool AT %DB5096.DBX16.5, 500 ms
   "2930RS001A01T01.DQ.SIG_OK" : Bool AT %DB5096.DBX16.6, 500 ms
   "2930RS001A01T01.DQ.LIM_H2" : Bool AT %DB5096.DBX16.7, 500 ms
   "2930RS001A01T01.DQ.LIM_H1" : Bool AT %DB5096.DBX17.0, 500 ms
   "2930RS001A01T01.DQ.LIM_L1" : Bool AT %DB5096.DBX17.1, 500 ms
   "2930RS001A01T01.DQ.LIM_L2" : Bool AT %DB5096.DBX17.2, 500 ms
   "2930RS001A01T01.DQ.GR_P" : Bool AT %DB5096.DBX17.3, 500 ms
   "2930RS001A01T01.DQ.GR_N" : Bool AT %DB5096.DBX17.4, 500 ms
   "2930RS001A01T01.I.IN" : Real AT %DB5096.DBD2, 500 ms
   "2930RS001A01T01.I.SIG_TYPE" : Int AT %DB5096.DBW0, 500 ms
   "2930RS001A01T01.I.FI_BUS" : Byte AT %DB5096.DBB6, 500 ms
   "2930RS001A01T01.DI.U_RANGE" : Bool AT %DB5096.DBX7.0, 500 ms
   "2930RS001A01T01.DI.O_RANGE" : Bool AT %DB5096.DBX7.1, 500 ms
   "2930RS001A01T01.DI.SIG_FAULT" : Bool AT %DB5096.DBX7.2, 500 ms
   "2930RS001A01T01.DI.EnConfig" : Bool AT %DB5096.DBX7.3, 500 ms
   "2930RS001A01T01.DI.AEN" : Bool AT %DB5096.DBX7.4, 500 ms
   "2930RS001A01T01.DI.AL_SUPR" : Bool AT %DB5096.DBX7.5, 500 ms
   "2930RS001A01T01.Q.PV_NORM" : Real AT %DB5096.DBD8, 500 ms
   "2930RS001A01T01.Q.PV_SCAL" : Real AT %DB5096.DBD12, 500 ms
   "2930RS001A01T01.ParentInfo" : TextRef, internal   // Имя родителя для попап окна, вкладка инфо. При експорте из ECS через скрипт заполняется автоматически, если теги копируются в ручную то требуется в ручную задатать свойство Start Value

HMI tags "2935RS001A01F01"
   "2935RS001A01F01.MSW" : 52809b66-421d-457f-8884-6f7a49d4e247 AT %DB5072.DBX18.0, 500 ms
   "2935RS001A01F01.DefaultText" : TextRef, internal   // Заголовок POPUP окна. При експорте из ECS через скрипт заполняется автоматически, если теги копируются в ручную то требуется в ручную задатать свойство Start Value
   "2935RS001A01F01.BlockInfo" : Array [0..2] of Int AT %DB5072.DBX38.0, 500 ms
   "2935RS001A01F01.StatusWork" : Int AT %DB5072.DBW242, 500 ms
   "2935RS001A01F01.FP_PARAM.DampingTime" : Int AT %DB5072.DBW50, 500 ms
   "2935RS001A01F01.FP_PARAM.Force_Value" : Real AT %DB5072.DBD52, 500 ms
   "2935RS001A01F01.FP_PARAM.Scale_Min" : Real AT %DB5072.DBD56, 500 ms
   "2935RS001A01F01.FP_PARAM.Scale_Max" : Real AT %DB5072.DBD60, 500 ms
   "2935RS001A01F01.FP_PARAM.Gradient" : Real AT %DB5072.DBD64, 500 ms
   "2935RS001A01F01.FP_PARAM.Grad_Pos" : Real AT %DB5072.DBD68, 500 ms
   "2935RS001A01F01.FP_PARAM.Grad_Neg" : Real AT %DB5072.DBD72, 500 ms
   "2935RS001A01F01.FP_PARAM.Grad_X" : Real AT %DB5072.DBD76, 500 ms
   "2935RS001A01F01.FP_PARAM.Gradient_Time_Pre" : Int AT %DB5072.DBW80, 500 ms
   "2935RS001A01F01.FP_PARAM.Gradient_Time_ACC" : Int AT %DB5072.DBW82, 500 ms
   "2935RS001A01F01.FP_PARAM.Alarm_Hyst" : Real AT %DB5072.DBD84, 500 ms
   "2935RS001A01F01.FP_PARAM.AlarmLimit_H3" : Real AT %DB5072.DBD88, 500 ms
   "2935RS001A01F01.FP_PARAM.AlarmLimit_H2" : Real AT %DB5072.DBD92, 500 ms
   "2935RS001A01F01.FP_PARAM.AlarmLimit_H1" : Real AT %DB5072.DBD96, 500 ms
   "2935RS001A01F01.FP_PARAM.AlarmLimit_L1" : Real AT %DB5072.DBD100, 500 ms
   "2935RS001A01F01.FP_PARAM.AlarmLimit_L2" : Real AT %DB5072.DBD104, 500 ms
   "2935RS001A01F01.FP_PARAM.AlarmLimit_L3" : Real AT %DB5072.DBD108, 500 ms
   "2935RS001A01F01.FP_PARAM.AlarmDelay_H3_Pre" : Int AT %DB5072.DBW112, 500 ms
   "2935RS001A01F01.FP_PARAM.AlarmDelay_H3_Acc" : Int AT %DB5072.DBW114, 500 ms
   "2935RS001A01F01.FP_PARAM.AlarmDelay_H2_Pre" : Int AT %DB5072.DBW116, 500 ms
   "2935RS001A01F01.FP_PARAM.AlarmDelay_H2_Acc" : Int AT %DB5072.DBW118, 500 ms
   "2935RS001A01F01.FP_PARAM.AlarmDelay_H1_Pre" : Int AT %DB5072.DBW120, 500 ms
   "2935RS001A01F01.FP_PARAM.AlarmDelay_H1_Acc" : Int AT %DB5072.DBW122, 500 ms
   "2935RS001A01F01.FP_PARAM.AlarmDelay_L1_Pre" : Int AT %DB5072.DBW124, 500 ms
   "2935RS001A01F01.FP_PARAM.AlarmDelay_L1_Acc" : Int AT %DB5072.DBW126, 500 ms
   "2935RS001A01F01.FP_PARAM.AlarmDelay_L2_Pre" : Int AT %DB5072.DBW128, 500 ms
   "2935RS001A01F01.FP_PARAM.AlarmDelay_L2_Acc" : Int AT %DB5072.DBW130, 500 ms
   "2935RS001A01F01.FP_PARAM.AlarmDelay_L3_Pre" : Int AT %DB5072.DBW132, 500 ms
   "2935RS001A01F01.FP_PARAM.AlarmDelay_L3_Acc" : Int AT %DB5072.DBW134, 500 ms
   "2935RS001A01F01.FP_PARAM.OpenLoopDelay_Pre" : Int AT %DB5072.DBW136, 500 ms
   "2935RS001A01F01.FP_PARAM.OpenLoopDelay_Acc" : Int AT %DB5072.DBW138, 500 ms
   "2935RS001A01F01.FP_PARAM.OverRangeDelay_Pre" : Int AT %DB5072.DBW140, 500 ms
   "2935RS001A01F01.FP_PARAM.OverRangeDelay_Acc" : Int AT %DB5072.DBW142, 500 ms
   "2935RS001A01F01.FP_PARAM.AuxLimit_H2_Value" : Real AT %DB5072.DBD144, 500 ms
   "2935RS001A01F01.FP_PARAM.AuxLimit_H1_Value" : Real AT %DB5072.DBD148, 500 ms
   "2935RS001A01F01.FP_PARAM.AuxLimit_L2_Value" : Real AT %DB5072.DBD152, 500 ms
   "2935RS001A01F01.FP_PARAM.AuxLimit_L1_Value" : Real AT %DB5072.DBD156, 500 ms
   "2935RS001A01F01.Unit" : TextRef, internal   // Еденицы измерения При експорте из ECS через скрипт заполняется автоматически, если теги копируются в ручную то требуется задатать свойство Text
   "2935RS001A01F01.Decimals" : TextRef, internal   // Формат отображения При експорте из ECS через скрипт, заполняется автоматически. Если теги копируются в ручную то требуется задатать свойство Text s999999.9
   "2935RS001A01F01.FP_EN.Square" : Bool AT %DB5072.DBX46.0, 500 ms
   "2935RS001A01F01.FP_EN.SquareRoot" : Bool AT %DB5072.DBX46.1, 500 ms
   "2935RS001A01F01.FP_EN.ParentSupress" : Bool AT %DB5072.DBX46.2, 500 ms
   "2935RS001A01F01.FP_EN.ParentSupressUnit" : Bool AT %DB5072.DBX46.3, 500 ms
   "2935RS001A01F01.FP_EN.Force" : Bool AT %DB5072.DBX46.4, 500 ms
   "2935RS001A01F01.FP_EN.Damping" : Bool AT %DB5072.DBX46.5, 500 ms
   "2935RS001A01F01.FP_EN.Gradient_Pos" : Bool AT %DB5072.DBX46.6, 500 ms
   "2935RS001A01F01.FP_EN.Gradient_Neg" : Bool AT %DB5072.DBX46.7, 500 ms
   "2935RS001A01F01.FP_EN.Hysteresis" : Bool AT %DB5072.DBX47.0, 500 ms
   "2935RS001A01F01.FP_EN.Alarm_H3" : Bool AT %DB5072.DBX47.1, 500 ms
   "2935RS001A01F01.FP_EN.Alarm_H2" : Bool AT %DB5072.DBX47.2, 500 ms
   "2935RS001A01F01.FP_EN.Alarm_H1" : Bool AT %DB5072.DBX47.3, 500 ms
   "2935RS001A01F01.FP_EN.Alarm_L1" : Bool AT %DB5072.DBX47.4, 500 ms
   "2935RS001A01F01.FP_EN.Alarm_L2" : Bool AT %DB5072.DBX47.5, 500 ms
   "2935RS001A01F01.FP_EN.Alarm_L3" : Bool AT %DB5072.DBX47.6, 500 ms
   "2935RS001A01F01.FP_EN.AlarmDelay_H3" : Bool AT %DB5072.DBX47.7, 500 ms
   "2935RS001A01F01.FP_EN.AlarmDelay_H2" : Bool AT %DB5072.DBX48.0, 500 ms
   "2935RS001A01F01.FP_EN.AlarmDelay_H1" : Bool AT %DB5072.DBX48.1, 500 ms
   "2935RS001A01F01.FP_EN.AlarmDelay_L1" : Bool AT %DB5072.DBX48.2, 500 ms
   "2935RS001A01F01.FP_EN.AlarmDelay_L2" : Bool AT %DB5072.DBX48.3, 500 ms
   "2935RS001A01F01.FP_EN.AlarmDelay_L3" : Bool AT %DB5072.DBX48.4, 500 ms
   "2935RS001A01F01.FP_EN.ROC_Warn" : Bool AT %DB5072.DBX48.5, 500 ms
   "2935RS001A01F01.FP_EN.U_Range_Warn" : Bool AT %DB5072.DBX48.6, 500 ms
   "2935RS001A01F01.FP_EN.O_Range_Warn" : Bool AT %DB5072.DBX48.7, 500 ms
   "2935RS001A01F01.trend_tag_name" : TextRef, internal   // Еденицы измерения При експорте из ECS через скрипт - заполняется автоматически, если теги копируются в ручную то требуется задатать свойство Text - имя тега для тренда
   "2935RS001A01F01.DQ.AL_H3" : Bool AT %DB5072.DBX16.0, 500 ms
   "2935RS001A01F01.DQ.AL_H2" : Bool AT %DB5072.DBX16.1, 500 ms
   "2935RS001A01F01.DQ.AL_H1" : Bool AT %DB5072.DBX16.2, 500 ms
   "2935RS001A01F01.DQ.AL_L1" : Bool AT %DB5072.DBX16.3, 500 ms
   "2935RS001A01F01.DQ.AL_L2" : Bool AT %DB5072.DBX16.4, 500 ms
   "2935RS001A01F01.DQ.AL_L3" : Bool AT %DB5072.DBX16.5, 500 ms
   "2935RS001A01F01.DQ.SIG_OK" : Bool AT %DB5072.DBX16.6, 500 ms
   "2935RS001A01F01.DQ.LIM_H2" : Bool AT %DB5072.DBX16.7, 500 ms
   "2935RS001A01F01.DQ.LIM_H1" : Bool AT %DB5072.DBX17.0, 500 ms
   "2935RS001A01F01.DQ.LIM_L1" : Bool AT %DB5072.DBX17.1, 500 ms
   "2935RS001A01F01.DQ.LIM_L2" : Bool AT %DB5072.DBX17.2, 500 ms
   "2935RS001A01F01.DQ.GR_P" : Bool AT %DB5072.DBX17.3, 500 ms
   "2935RS001A01F01.DQ.GR_N" : Bool AT %DB5072.DBX17.4, 500 ms
   "2935RS001A01F01.I.IN" : Real AT %DB5072.DBD2, 500 ms
   "2935RS001A01F01.I.SIG_TYPE" : Int AT %DB5072.DBW0, 500 ms
   "2935RS001A01F01.I.FI_BUS" : Byte AT %DB5072.DBB6, 500 ms
   "2935RS001A01F01.DI.U_RANGE" : Bool AT %DB5072.DBX7.0, 500 ms
   "2935RS001A01F01.DI.O_RANGE" : Bool AT %DB5072.DBX7.1, 500 ms
   "2935RS001A01F01.DI.SIG_FAULT" : Bool AT %DB5072.DBX7.2, 500 ms
   "2935RS001A01F01.DI.EnConfig" : Bool AT %DB5072.DBX7.3, 500 ms
   "2935RS001A01F01.DI.AEN" : Bool AT %DB5072.DBX7.4, 500 ms
   "2935RS001A01F01.DI.AL_SUPR" : Bool AT %DB5072.DBX7.5, 500 ms
   "2935RS001A01F01.Q.PV_NORM" : Real AT %DB5072.DBD8, 500 ms
   "2935RS001A01F01.Q.PV_SCAL" : Real AT %DB5072.DBD12, 500 ms
   "2935RS001A01F01.ParentInfo" : TextRef, internal   // Имя родителя для попап окна, вкладка инфо. При експорте из ECS через скрипт заполняется автоматически, если теги копируются в ручную то требуется в ручную задатать свойство Start Value

HMI tags "2935RS001A01F02"
   "2935RS001A01F02.MSW" : 52809b66-421d-457f-8884-6f7a49d4e247 AT %DB5073.DBX18.0, 500 ms
   "2935RS001A01F02.DefaultText" : TextRef, internal   // Заголовок POPUP окна. При експорте из ECS через скрипт заполняется автоматически, если теги копируются в ручную то требуется в ручную задатать свойство Start Value
   "2935RS001A01F02.BlockInfo" : Array [0..2] of Int AT %DB5073.DBX38.0, 500 ms
   "2935RS001A01F02.StatusWork" : Int AT %DB5073.DBW242, 500 ms
   "2935RS001A01F02.FP_PARAM.DampingTime" : Int AT %DB5073.DBW50, 500 ms
   "2935RS001A01F02.FP_PARAM.Force_Value" : Real AT %DB5073.DBD52, 500 ms
   "2935RS001A01F02.FP_PARAM.Scale_Min" : Real AT %DB5073.DBD56, 500 ms
   "2935RS001A01F02.FP_PARAM.Scale_Max" : Real AT %DB5073.DBD60, 500 ms
   "2935RS001A01F02.FP_PARAM.Gradient" : Real AT %DB5073.DBD64, 500 ms
   "2935RS001A01F02.FP_PARAM.Grad_Pos" : Real AT %DB5073.DBD68, 500 ms
   "2935RS001A01F02.FP_PARAM.Grad_Neg" : Real AT %DB5073.DBD72, 500 ms
   "2935RS001A01F02.FP_PARAM.Grad_X" : Real AT %DB5073.DBD76, 500 ms
   "2935RS001A01F02.FP_PARAM.Gradient_Time_Pre" : Int AT %DB5073.DBW80, 500 ms
   "2935RS001A01F02.FP_PARAM.Gradient_Time_ACC" : Int AT %DB5073.DBW82, 500 ms
   "2935RS001A01F02.FP_PARAM.Alarm_Hyst" : Real AT %DB5073.DBD84, 500 ms
   "2935RS001A01F02.FP_PARAM.AlarmLimit_H3" : Real AT %DB5073.DBD88, 500 ms
   "2935RS001A01F02.FP_PARAM.AlarmLimit_H2" : Real AT %DB5073.DBD92, 500 ms
   "2935RS001A01F02.FP_PARAM.AlarmLimit_H1" : Real AT %DB5073.DBD96, 500 ms
   "2935RS001A01F02.FP_PARAM.AlarmLimit_L1" : Real AT %DB5073.DBD100, 500 ms
   "2935RS001A01F02.FP_PARAM.AlarmLimit_L2" : Real AT %DB5073.DBD104, 500 ms
   "2935RS001A01F02.FP_PARAM.AlarmLimit_L3" : Real AT %DB5073.DBD108, 500 ms
   "2935RS001A01F02.FP_PARAM.AlarmDelay_H3_Pre" : Int AT %DB5073.DBW112, 500 ms
   "2935RS001A01F02.FP_PARAM.AlarmDelay_H3_Acc" : Int AT %DB5073.DBW114, 500 ms
   "2935RS001A01F02.FP_PARAM.AlarmDelay_H2_Pre" : Int AT %DB5073.DBW116, 500 ms
   "2935RS001A01F02.FP_PARAM.AlarmDelay_H2_Acc" : Int AT %DB5073.DBW118, 500 ms
   "2935RS001A01F02.FP_PARAM.AlarmDelay_H1_Pre" : Int AT %DB5073.DBW120, 500 ms
   "2935RS001A01F02.FP_PARAM.AlarmDelay_H1_Acc" : Int AT %DB5073.DBW122, 500 ms
   "2935RS001A01F02.FP_PARAM.AlarmDelay_L1_Pre" : Int AT %DB5073.DBW124, 500 ms
   "2935RS001A01F02.FP_PARAM.AlarmDelay_L1_Acc" : Int AT %DB5073.DBW126, 500 ms
   "2935RS001A01F02.FP_PARAM.AlarmDelay_L2_Pre" : Int AT %DB5073.DBW128, 500 ms
   "2935RS001A01F02.FP_PARAM.AlarmDelay_L2_Acc" : Int AT %DB5073.DBW130, 500 ms
   "2935RS001A01F02.FP_PARAM.AlarmDelay_L3_Pre" : Int AT %DB5073.DBW132, 500 ms
   "2935RS001A01F02.FP_PARAM.AlarmDelay_L3_Acc" : Int AT %DB5073.DBW134, 500 ms
   "2935RS001A01F02.FP_PARAM.OpenLoopDelay_Pre" : Int AT %DB5073.DBW136, 500 ms
   "2935RS001A01F02.FP_PARAM.OpenLoopDelay_Acc" : Int AT %DB5073.DBW138, 500 ms
   "2935RS001A01F02.FP_PARAM.OverRangeDelay_Pre" : Int AT %DB5073.DBW140, 500 ms
   "2935RS001A01F02.FP_PARAM.OverRangeDelay_Acc" : Int AT %DB5073.DBW142, 500 ms
   "2935RS001A01F02.FP_PARAM.AuxLimit_H2_Value" : Real AT %DB5073.DBD144, 500 ms
   "2935RS001A01F02.FP_PARAM.AuxLimit_H1_Value" : Real AT %DB5073.DBD148, 500 ms
   "2935RS001A01F02.FP_PARAM.AuxLimit_L2_Value" : Real AT %DB5073.DBD152, 500 ms
   "2935RS001A01F02.FP_PARAM.AuxLimit_L1_Value" : Real AT %DB5073.DBD156, 500 ms
   "2935RS001A01F02.Unit" : TextRef, internal   // Еденицы измерения При експорте из ECS через скрипт заполняется автоматически, если теги копируются в ручную то требуется задатать свойство Text
   "2935RS001A01F02.Decimals" : TextRef, internal   // Формат отображения При експорте из ECS через скрипт, заполняется автоматически. Если теги копируются в ручную то требуется задатать свойство Text s999999.9
   "2935RS001A01F02.FP_EN.Square" : Bool AT %DB5073.DBX46.0, 500 ms
   "2935RS001A01F02.FP_EN.SquareRoot" : Bool AT %DB5073.DBX46.1, 500 ms
   "2935RS001A01F02.FP_EN.ParentSupress" : Bool AT %DB5073.DBX46.2, 500 ms
   "2935RS001A01F02.FP_EN.ParentSupressUnit" : Bool AT %DB5073.DBX46.3, 500 ms
   "2935RS001A01F02.FP_EN.Force" : Bool AT %DB5073.DBX46.4, 500 ms
   "2935RS001A01F02.FP_EN.Damping" : Bool AT %DB5073.DBX46.5, 500 ms
   "2935RS001A01F02.FP_EN.Gradient_Pos" : Bool AT %DB5073.DBX46.6, 500 ms
   "2935RS001A01F02.FP_EN.Gradient_Neg" : Bool AT %DB5073.DBX46.7, 500 ms
   "2935RS001A01F02.FP_EN.Hysteresis" : Bool AT %DB5073.DBX47.0, 500 ms
   "2935RS001A01F02.FP_EN.Alarm_H3" : Bool AT %DB5073.DBX47.1, 500 ms
   "2935RS001A01F02.FP_EN.Alarm_H2" : Bool AT %DB5073.DBX47.2, 500 ms
   "2935RS001A01F02.FP_EN.Alarm_H1" : Bool AT %DB5073.DBX47.3, 500 ms
   "2935RS001A01F02.FP_EN.Alarm_L1" : Bool AT %DB5073.DBX47.4, 500 ms
   "2935RS001A01F02.FP_EN.Alarm_L2" : Bool AT %DB5073.DBX47.5, 500 ms
   "2935RS001A01F02.FP_EN.Alarm_L3" : Bool AT %DB5073.DBX47.6, 500 ms
   "2935RS001A01F02.FP_EN.AlarmDelay_H3" : Bool AT %DB5073.DBX47.7, 500 ms
   "2935RS001A01F02.FP_EN.AlarmDelay_H2" : Bool AT %DB5073.DBX48.0, 500 ms
   "2935RS001A01F02.FP_EN.AlarmDelay_H1" : Bool AT %DB5073.DBX48.1, 500 ms
   "2935RS001A01F02.FP_EN.AlarmDelay_L1" : Bool AT %DB5073.DBX48.2, 500 ms
   "2935RS001A01F02.FP_EN.AlarmDelay_L2" : Bool AT %DB5073.DBX48.3, 500 ms
   "2935RS001A01F02.FP_EN.AlarmDelay_L3" : Bool AT %DB5073.DBX48.4, 500 ms
   "2935RS001A01F02.FP_EN.ROC_Warn" : Bool AT %DB5073.DBX48.5, 500 ms
   "2935RS001A01F02.FP_EN.U_Range_Warn" : Bool AT %DB5073.DBX48.6, 500 ms
   "2935RS001A01F02.FP_EN.O_Range_Warn" : Bool AT %DB5073.DBX48.7, 500 ms
   "2935RS001A01F02.trend_tag_name" : TextRef, internal   // Еденицы измерения При експорте из ECS через скрипт - заполняется автоматически, если теги копируются в ручную то требуется задатать свойство Text - имя тега для тренда
   "2935RS001A01F02.DQ.AL_H3" : Bool AT %DB5073.DBX16.0, 500 ms
   "2935RS001A01F02.DQ.AL_H2" : Bool AT %DB5073.DBX16.1, 500 ms
   "2935RS001A01F02.DQ.AL_H1" : Bool AT %DB5073.DBX16.2, 500 ms
   "2935RS001A01F02.DQ.AL_L1" : Bool AT %DB5073.DBX16.3, 500 ms
   "2935RS001A01F02.DQ.AL_L2" : Bool AT %DB5073.DBX16.4, 500 ms
   "2935RS001A01F02.DQ.AL_L3" : Bool AT %DB5073.DBX16.5, 500 ms
   "2935RS001A01F02.DQ.SIG_OK" : Bool AT %DB5073.DBX16.6, 500 ms
   "2935RS001A01F02.DQ.LIM_H2" : Bool AT %DB5073.DBX16.7, 500 ms
   "2935RS001A01F02.DQ.LIM_H1" : Bool AT %DB5073.DBX17.0, 500 ms
   "2935RS001A01F02.DQ.LIM_L1" : Bool AT %DB5073.DBX17.1, 500 ms
   "2935RS001A01F02.DQ.LIM_L2" : Bool AT %DB5073.DBX17.2, 500 ms
   "2935RS001A01F02.DQ.GR_P" : Bool AT %DB5073.DBX17.3, 500 ms
   "2935RS001A01F02.DQ.GR_N" : Bool AT %DB5073.DBX17.4, 500 ms
   "2935RS001A01F02.I.IN" : Real AT %DB5073.DBD2, 500 ms
   "2935RS001A01F02.I.SIG_TYPE" : Int AT %DB5073.DBW0, 500 ms
   "2935RS001A01F02.I.FI_BUS" : Byte AT %DB5073.DBB6, 500 ms
   "2935RS001A01F02.DI.U_RANGE" : Bool AT %DB5073.DBX7.0, 500 ms
   "2935RS001A01F02.DI.O_RANGE" : Bool AT %DB5073.DBX7.1, 500 ms
   "2935RS001A01F02.DI.SIG_FAULT" : Bool AT %DB5073.DBX7.2, 500 ms
   "2935RS001A01F02.DI.EnConfig" : Bool AT %DB5073.DBX7.3, 500 ms
   "2935RS001A01F02.DI.AEN" : Bool AT %DB5073.DBX7.4, 500 ms
   "2935RS001A01F02.DI.AL_SUPR" : Bool AT %DB5073.DBX7.5, 500 ms
   "2935RS001A01F02.Q.PV_NORM" : Real AT %DB5073.DBD8, 500 ms
   "2935RS001A01F02.Q.PV_SCAL" : Real AT %DB5073.DBD12, 500 ms
   "2935RS001A01F02.ParentInfo" : TextRef, internal   // Имя родителя для попап окна, вкладка инфо. При експорте из ECS через скрипт заполняется автоматически, если теги копируются в ручную то требуется в ручную задатать свойство Start Value

HMI tags "2935RS001A01F03"
   "2935RS001A01F03.MSW" : 52809b66-421d-457f-8884-6f7a49d4e247 AT %DB5074.DBX18.0, 500 ms
   "2935RS001A01F03.DefaultText" : TextRef, internal   // Заголовок POPUP окна. При експорте из ECS через скрипт заполняется автоматически, если теги копируются в ручную то требуется в ручную задатать свойство Start Value
   "2935RS001A01F03.BlockInfo" : Array [0..2] of Int AT %DB5074.DBX38.0, 500 ms
   "2935RS001A01F03.StatusWork" : Int AT %DB5074.DBW242, 500 ms
   "2935RS001A01F03.FP_PARAM.DampingTime" : Int AT %DB5074.DBW50, 500 ms
   "2935RS001A01F03.FP_PARAM.Force_Value" : Real AT %DB5074.DBD52, 500 ms
   "2935RS001A01F03.FP_PARAM.Scale_Min" : Real AT %DB5074.DBD56, 500 ms
   "2935RS001A01F03.FP_PARAM.Scale_Max" : Real AT %DB5074.DBD60, 500 ms
   "2935RS001A01F03.FP_PARAM.Gradient" : Real AT %DB5074.DBD64, 500 ms
   "2935RS001A01F03.FP_PARAM.Grad_Pos" : Real AT %DB5074.DBD68, 500 ms
   "2935RS001A01F03.FP_PARAM.Grad_Neg" : Real AT %DB5074.DBD72, 500 ms
   "2935RS001A01F03.FP_PARAM.Grad_X" : Real AT %DB5074.DBD76, 500 ms
   "2935RS001A01F03.FP_PARAM.Gradient_Time_Pre" : Int AT %DB5074.DBW80, 500 ms
   "2935RS001A01F03.FP_PARAM.Gradient_Time_ACC" : Int AT %DB5074.DBW82, 500 ms
   "2935RS001A01F03.FP_PARAM.Alarm_Hyst" : Real AT %DB5074.DBD84, 500 ms
   "2935RS001A01F03.FP_PARAM.AlarmLimit_H3" : Real AT %DB5074.DBD88, 500 ms
   "2935RS001A01F03.FP_PARAM.AlarmLimit_H2" : Real AT %DB5074.DBD92, 500 ms
   "2935RS001A01F03.FP_PARAM.AlarmLimit_H1" : Real AT %DB5074.DBD96, 500 ms
   "2935RS001A01F03.FP_PARAM.AlarmLimit_L1" : Real AT %DB5074.DBD100, 500 ms
   "2935RS001A01F03.FP_PARAM.AlarmLimit_L2" : Real AT %DB5074.DBD104, 500 ms
   "2935RS001A01F03.FP_PARAM.AlarmLimit_L3" : Real AT %DB5074.DBD108, 500 ms
   "2935RS001A01F03.FP_PARAM.AlarmDelay_H3_Pre" : Int AT %DB5074.DBW112, 500 ms
   "2935RS001A01F03.FP_PARAM.AlarmDelay_H3_Acc" : Int AT %DB5074.DBW114, 500 ms
   "2935RS001A01F03.FP_PARAM.AlarmDelay_H2_Pre" : Int AT %DB5074.DBW116, 500 ms
   "2935RS001A01F03.FP_PARAM.AlarmDelay_H2_Acc" : Int AT %DB5074.DBW118, 500 ms
   "2935RS001A01F03.FP_PARAM.AlarmDelay_H1_Pre" : Int AT %DB5074.DBW120, 500 ms
   "2935RS001A01F03.FP_PARAM.AlarmDelay_H1_Acc" : Int AT %DB5074.DBW122, 500 ms
   "2935RS001A01F03.FP_PARAM.AlarmDelay_L1_Pre" : Int AT %DB5074.DBW124, 500 ms
   "2935RS001A01F03.FP_PARAM.AlarmDelay_L1_Acc" : Int AT %DB5074.DBW126, 500 ms
   "2935RS001A01F03.FP_PARAM.AlarmDelay_L2_Pre" : Int AT %DB5074.DBW128, 500 ms
   "2935RS001A01F03.FP_PARAM.AlarmDelay_L2_Acc" : Int AT %DB5074.DBW130, 500 ms
   "2935RS001A01F03.FP_PARAM.AlarmDelay_L3_Pre" : Int AT %DB5074.DBW132, 500 ms
   "2935RS001A01F03.FP_PARAM.AlarmDelay_L3_Acc" : Int AT %DB5074.DBW134, 500 ms
   "2935RS001A01F03.FP_PARAM.OpenLoopDelay_Pre" : Int AT %DB5074.DBW136, 500 ms
   "2935RS001A01F03.FP_PARAM.OpenLoopDelay_Acc" : Int AT %DB5074.DBW138, 500 ms
   "2935RS001A01F03.FP_PARAM.OverRangeDelay_Pre" : Int AT %DB5074.DBW140, 500 ms
   "2935RS001A01F03.FP_PARAM.OverRangeDelay_Acc" : Int AT %DB5074.DBW142, 500 ms
   "2935RS001A01F03.FP_PARAM.AuxLimit_H2_Value" : Real AT %DB5074.DBD144, 500 ms
   "2935RS001A01F03.FP_PARAM.AuxLimit_H1_Value" : Real AT %DB5074.DBD148, 500 ms
   "2935RS001A01F03.FP_PARAM.AuxLimit_L2_Value" : Real AT %DB5074.DBD152, 500 ms
   "2935RS001A01F03.FP_PARAM.AuxLimit_L1_Value" : Real AT %DB5074.DBD156, 500 ms
   "2935RS001A01F03.Unit" : TextRef, internal   // Еденицы измерения При експорте из ECS через скрипт заполняется автоматически, если теги копируются в ручную то требуется задатать свойство Text
   "2935RS001A01F03.Decimals" : TextRef, internal   // Формат отображения При експорте из ECS через скрипт, заполняется автоматически. Если теги копируются в ручную то требуется задатать свойство Text s999999.9
   "2935RS001A01F03.FP_EN.Square" : Bool AT %DB5074.DBX46.0, 500 ms
   "2935RS001A01F03.FP_EN.SquareRoot" : Bool AT %DB5074.DBX46.1, 500 ms
   "2935RS001A01F03.FP_EN.ParentSupress" : Bool AT %DB5074.DBX46.2, 500 ms
   "2935RS001A01F03.FP_EN.ParentSupressUnit" : Bool AT %DB5074.DBX46.3, 500 ms
   "2935RS001A01F03.FP_EN.Force" : Bool AT %DB5074.DBX46.4, 500 ms
   "2935RS001A01F03.FP_EN.Damping" : Bool AT %DB5074.DBX46.5, 500 ms
   "2935RS001A01F03.FP_EN.Gradient_Pos" : Bool AT %DB5074.DBX46.6, 500 ms
   "2935RS001A01F03.FP_EN.Gradient_Neg" : Bool AT %DB5074.DBX46.7, 500 ms
   "2935RS001A01F03.FP_EN.Hysteresis" : Bool AT %DB5074.DBX47.0, 500 ms
   "2935RS001A01F03.FP_EN.Alarm_H3" : Bool AT %DB5074.DBX47.1, 500 ms
   "2935RS001A01F03.FP_EN.Alarm_H2" : Bool AT %DB5074.DBX47.2, 500 ms
   "2935RS001A01F03.FP_EN.Alarm_H1" : Bool AT %DB5074.DBX47.3, 500 ms
   "2935RS001A01F03.FP_EN.Alarm_L1" : Bool AT %DB5074.DBX47.4, 500 ms
   "2935RS001A01F03.FP_EN.Alarm_L2" : Bool AT %DB5074.DBX47.5, 500 ms
   "2935RS001A01F03.FP_EN.Alarm_L3" : Bool AT %DB5074.DBX47.6, 500 ms
   "2935RS001A01F03.FP_EN.AlarmDelay_H3" : Bool AT %DB5074.DBX47.7, 500 ms
   "2935RS001A01F03.FP_EN.AlarmDelay_H2" : Bool AT %DB5074.DBX48.0, 500 ms
   "2935RS001A01F03.FP_EN.AlarmDelay_H1" : Bool AT %DB5074.DBX48.1, 500 ms
   "2935RS001A01F03.FP_EN.AlarmDelay_L1" : Bool AT %DB5074.DBX48.2, 500 ms
   "2935RS001A01F03.FP_EN.AlarmDelay_L2" : Bool AT %DB5074.DBX48.3, 500 ms
   "2935RS001A01F03.FP_EN.AlarmDelay_L3" : Bool AT %DB5074.DBX48.4, 500 ms
   "2935RS001A01F03.FP_EN.ROC_Warn" : Bool AT %DB5074.DBX48.5, 500 ms
   "2935RS001A01F03.FP_EN.U_Range_Warn" : Bool AT %DB5074.DBX48.6, 500 ms
   "2935RS001A01F03.FP_EN.O_Range_Warn" : Bool AT %DB5074.DBX48.7, 500 ms
   "2935RS001A01F03.trend_tag_name" : TextRef, internal   // Еденицы измерения При експорте из ECS через скрипт - заполняется автоматически, если теги копируются в ручную то требуется задатать свойство Text - имя тега для тренда
   "2935RS001A01F03.DQ.AL_H3" : Bool AT %DB5074.DBX16.0, 500 ms
   "2935RS001A01F03.DQ.AL_H2" : Bool AT %DB5074.DBX16.1, 500 ms
   "2935RS001A01F03.DQ.AL_H1" : Bool AT %DB5074.DBX16.2, 500 ms
   "2935RS001A01F03.DQ.AL_L1" : Bool AT %DB5074.DBX16.3, 500 ms
   "2935RS001A01F03.DQ.AL_L2" : Bool AT %DB5074.DBX16.4, 500 ms
   "2935RS001A01F03.DQ.AL_L3" : Bool AT %DB5074.DBX16.5, 500 ms
   "2935RS001A01F03.DQ.SIG_OK" : Bool AT %DB5074.DBX16.6, 500 ms
   "2935RS001A01F03.DQ.LIM_H2" : Bool AT %DB5074.DBX16.7, 500 ms
   "2935RS001A01F03.DQ.LIM_H1" : Bool AT %DB5074.DBX17.0, 500 ms
   "2935RS001A01F03.DQ.LIM_L1" : Bool AT %DB5074.DBX17.1, 500 ms
   "2935RS001A01F03.DQ.LIM_L2" : Bool AT %DB5074.DBX17.2, 500 ms
   "2935RS001A01F03.DQ.GR_P" : Bool AT %DB5074.DBX17.3, 500 ms
   "2935RS001A01F03.DQ.GR_N" : Bool AT %DB5074.DBX17.4, 500 ms
   "2935RS001A01F03.I.IN" : Real AT %DB5074.DBD2, 500 ms
   "2935RS001A01F03.I.SIG_TYPE" : Int AT %DB5074.DBW0, 500 ms
   "2935RS001A01F03.I.FI_BUS" : Byte AT %DB5074.DBB6, 500 ms
   "2935RS001A01F03.DI.U_RANGE" : Bool AT %DB5074.DBX7.0, 500 ms
   "2935RS001A01F03.DI.O_RANGE" : Bool AT %DB5074.DBX7.1, 500 ms
   "2935RS001A01F03.DI.SIG_FAULT" : Bool AT %DB5074.DBX7.2, 500 ms
   "2935RS001A01F03.DI.EnConfig" : Bool AT %DB5074.DBX7.3, 500 ms
   "2935RS001A01F03.DI.AEN" : Bool AT %DB5074.DBX7.4, 500 ms
   "2935RS001A01F03.DI.AL_SUPR" : Bool AT %DB5074.DBX7.5, 500 ms
   "2935RS001A01F03.Q.PV_NORM" : Real AT %DB5074.DBD8, 500 ms
   "2935RS001A01F03.Q.PV_SCAL" : Real AT %DB5074.DBD12, 500 ms
   "2935RS001A01F03.ParentInfo" : TextRef, internal   // Имя родителя для попап окна, вкладка инфо. При експорте из ECS через скрипт заполняется автоматически, если теги копируются в ручную то требуется в ручную задатать свойство Start Value

HMI tags "2935RS001A01L01"
   "2935RS001A01L01.MSW" : 52809b66-421d-457f-8884-6f7a49d4e247 AT %DB5075.DBX18.0, 500 ms
   "2935RS001A01L01.DefaultText" : TextRef, internal   // Заголовок POPUP окна. При експорте из ECS через скрипт заполняется автоматически, если теги копируются в ручную то требуется в ручную задатать свойство Start Value
   "2935RS001A01L01.BlockInfo" : Array [0..2] of Int AT %DB5075.DBX38.0, 500 ms
   "2935RS001A01L01.StatusWork" : Int AT %DB5075.DBW242, 500 ms
   "2935RS001A01L01.FP_PARAM.DampingTime" : Int AT %DB5075.DBW50, 500 ms
   "2935RS001A01L01.FP_PARAM.Force_Value" : Real AT %DB5075.DBD52, 500 ms
   "2935RS001A01L01.FP_PARAM.Scale_Min" : Real AT %DB5075.DBD56, 500 ms
   "2935RS001A01L01.FP_PARAM.Scale_Max" : Real AT %DB5075.DBD60, 500 ms
   "2935RS001A01L01.FP_PARAM.Gradient" : Real AT %DB5075.DBD64, 500 ms
   "2935RS001A01L01.FP_PARAM.Grad_Pos" : Real AT %DB5075.DBD68, 500 ms
   "2935RS001A01L01.FP_PARAM.Grad_Neg" : Real AT %DB5075.DBD72, 500 ms
   "2935RS001A01L01.FP_PARAM.Grad_X" : Real AT %DB5075.DBD76, 500 ms
   "2935RS001A01L01.FP_PARAM.Gradient_Time_Pre" : Int AT %DB5075.DBW80, 500 ms
   "2935RS001A01L01.FP_PARAM.Gradient_Time_ACC" : Int AT %DB5075.DBW82, 500 ms
   "2935RS001A01L01.FP_PARAM.Alarm_Hyst" : Real AT %DB5075.DBD84, 500 ms
   "2935RS001A01L01.FP_PARAM.AlarmLimit_H3" : Real AT %DB5075.DBD88, 500 ms
   "2935RS001A01L01.FP_PARAM.AlarmLimit_H2" : Real AT %DB5075.DBD92, 500 ms
   "2935RS001A01L01.FP_PARAM.AlarmLimit_H1" : Real AT %DB5075.DBD96, 500 ms
   "2935RS001A01L01.FP_PARAM.AlarmLimit_L1" : Real AT %DB5075.DBD100, 500 ms
   "2935RS001A01L01.FP_PARAM.AlarmLimit_L2" : Real AT %DB5075.DBD104, 500 ms
   "2935RS001A01L01.FP_PARAM.AlarmLimit_L3" : Real AT %DB5075.DBD108, 500 ms
   "2935RS001A01L01.FP_PARAM.AlarmDelay_H3_Pre" : Int AT %DB5075.DBW112, 500 ms
   "2935RS001A01L01.FP_PARAM.AlarmDelay_H3_Acc" : Int AT %DB5075.DBW114, 500 ms
   "2935RS001A01L01.FP_PARAM.AlarmDelay_H2_Pre" : Int AT %DB5075.DBW116, 500 ms
   "2935RS001A01L01.FP_PARAM.AlarmDelay_H2_Acc" : Int AT %DB5075.DBW118, 500 ms
   "2935RS001A01L01.FP_PARAM.AlarmDelay_H1_Pre" : Int AT %DB5075.DBW120, 500 ms
   "2935RS001A01L01.FP_PARAM.AlarmDelay_H1_Acc" : Int AT %DB5075.DBW122, 500 ms
   "2935RS001A01L01.FP_PARAM.AlarmDelay_L1_Pre" : Int AT %DB5075.DBW124, 500 ms
   "2935RS001A01L01.FP_PARAM.AlarmDelay_L1_Acc" : Int AT %DB5075.DBW126, 500 ms
   "2935RS001A01L01.FP_PARAM.AlarmDelay_L2_Pre" : Int AT %DB5075.DBW128, 500 ms
   "2935RS001A01L01.FP_PARAM.AlarmDelay_L2_Acc" : Int AT %DB5075.DBW130, 500 ms
   "2935RS001A01L01.FP_PARAM.AlarmDelay_L3_Pre" : Int AT %DB5075.DBW132, 500 ms
   "2935RS001A01L01.FP_PARAM.AlarmDelay_L3_Acc" : Int AT %DB5075.DBW134, 500 ms
   "2935RS001A01L01.FP_PARAM.OpenLoopDelay_Pre" : Int AT %DB5075.DBW136, 500 ms
   "2935RS001A01L01.FP_PARAM.OpenLoopDelay_Acc" : Int AT %DB5075.DBW138, 500 ms
   "2935RS001A01L01.FP_PARAM.OverRangeDelay_Pre" : Int AT %DB5075.DBW140, 500 ms
   "2935RS001A01L01.FP_PARAM.OverRangeDelay_Acc" : Int AT %DB5075.DBW142, 500 ms
   "2935RS001A01L01.FP_PARAM.AuxLimit_H2_Value" : Real AT %DB5075.DBD144, 500 ms
   "2935RS001A01L01.FP_PARAM.AuxLimit_H1_Value" : Real AT %DB5075.DBD148, 500 ms
   "2935RS001A01L01.FP_PARAM.AuxLimit_L2_Value" : Real AT %DB5075.DBD152, 500 ms
   "2935RS001A01L01.FP_PARAM.AuxLimit_L1_Value" : Real AT %DB5075.DBD156, 500 ms
   "2935RS001A01L01.Unit" : TextRef, internal   // Еденицы измерения При експорте из ECS через скрипт заполняется автоматически, если теги копируются в ручную то требуется задатать свойство Text
   "2935RS001A01L01.Decimals" : TextRef, internal   // Формат отображения При експорте из ECS через скрипт, заполняется автоматически. Если теги копируются в ручную то требуется задатать свойство Text s999999.9
   "2935RS001A01L01.FP_EN.Square" : Bool AT %DB5075.DBX46.0, 500 ms
   "2935RS001A01L01.FP_EN.SquareRoot" : Bool AT %DB5075.DBX46.1, 500 ms
   "2935RS001A01L01.FP_EN.ParentSupress" : Bool AT %DB5075.DBX46.2, 500 ms
   "2935RS001A01L01.FP_EN.ParentSupressUnit" : Bool AT %DB5075.DBX46.3, 500 ms
   "2935RS001A01L01.FP_EN.Force" : Bool AT %DB5075.DBX46.4, 500 ms
   "2935RS001A01L01.FP_EN.Damping" : Bool AT %DB5075.DBX46.5, 500 ms
   "2935RS001A01L01.FP_EN.Gradient_Pos" : Bool AT %DB5075.DBX46.6, 500 ms
   "2935RS001A01L01.FP_EN.Gradient_Neg" : Bool AT %DB5075.DBX46.7, 500 ms
   "2935RS001A01L01.FP_EN.Hysteresis" : Bool AT %DB5075.DBX47.0, 500 ms
   "2935RS001A01L01.FP_EN.Alarm_H3" : Bool AT %DB5075.DBX47.1, 500 ms
   "2935RS001A01L01.FP_EN.Alarm_H2" : Bool AT %DB5075.DBX47.2, 500 ms
   "2935RS001A01L01.FP_EN.Alarm_H1" : Bool AT %DB5075.DBX47.3, 500 ms
   "2935RS001A01L01.FP_EN.Alarm_L1" : Bool AT %DB5075.DBX47.4, 500 ms
   "2935RS001A01L01.FP_EN.Alarm_L2" : Bool AT %DB5075.DBX47.5, 500 ms
   "2935RS001A01L01.FP_EN.Alarm_L3" : Bool AT %DB5075.DBX47.6, 500 ms
   "2935RS001A01L01.FP_EN.AlarmDelay_H3" : Bool AT %DB5075.DBX47.7, 500 ms
   "2935RS001A01L01.FP_EN.AlarmDelay_H2" : Bool AT %DB5075.DBX48.0, 500 ms
   "2935RS001A01L01.FP_EN.AlarmDelay_H1" : Bool AT %DB5075.DBX48.1, 500 ms
   "2935RS001A01L01.FP_EN.AlarmDelay_L1" : Bool AT %DB5075.DBX48.2, 500 ms
   "2935RS001A01L01.FP_EN.AlarmDelay_L2" : Bool AT %DB5075.DBX48.3, 500 ms
   "2935RS001A01L01.FP_EN.AlarmDelay_L3" : Bool AT %DB5075.DBX48.4, 500 ms
   "2935RS001A01L01.FP_EN.ROC_Warn" : Bool AT %DB5075.DBX48.5, 500 ms
   "2935RS001A01L01.FP_EN.U_Range_Warn" : Bool AT %DB5075.DBX48.6, 500 ms
   "2935RS001A01L01.FP_EN.O_Range_Warn" : Bool AT %DB5075.DBX48.7, 500 ms
   "2935RS001A01L01.trend_tag_name" : TextRef, internal   // Еденицы измерения При експорте из ECS через скрипт - заполняется автоматически, если теги копируются в ручную то требуется задатать свойство Text - имя тега для тренда
   "2935RS001A01L01.DQ.AL_H3" : Bool AT %DB5075.DBX16.0, 500 ms
   "2935RS001A01L01.DQ.AL_H2" : Bool AT %DB5075.DBX16.1, 500 ms
   "2935RS001A01L01.DQ.AL_H1" : Bool AT %DB5075.DBX16.2, 500 ms
   "2935RS001A01L01.DQ.AL_L1" : Bool AT %DB5075.DBX16.3, 500 ms
   "2935RS001A01L01.DQ.AL_L2" : Bool AT %DB5075.DBX16.4, 500 ms
   "2935RS001A01L01.DQ.AL_L3" : Bool AT %DB5075.DBX16.5, 500 ms
   "2935RS001A01L01.DQ.SIG_OK" : Bool AT %DB5075.DBX16.6, 500 ms
   "2935RS001A01L01.DQ.LIM_H2" : Bool AT %DB5075.DBX16.7, 500 ms
   "2935RS001A01L01.DQ.LIM_H1" : Bool AT %DB5075.DBX17.0, 500 ms
   "2935RS001A01L01.DQ.LIM_L1" : Bool AT %DB5075.DBX17.1, 500 ms
   "2935RS001A01L01.DQ.LIM_L2" : Bool AT %DB5075.DBX17.2, 500 ms
   "2935RS001A01L01.DQ.GR_P" : Bool AT %DB5075.DBX17.3, 500 ms
   "2935RS001A01L01.DQ.GR_N" : Bool AT %DB5075.DBX17.4, 500 ms
   "2935RS001A01L01.I.IN" : Real AT %DB5075.DBD2, 500 ms
   "2935RS001A01L01.I.SIG_TYPE" : Int AT %DB5075.DBW0, 500 ms
   "2935RS001A01L01.I.FI_BUS" : Byte AT %DB5075.DBB6, 500 ms
   "2935RS001A01L01.DI.U_RANGE" : Bool AT %DB5075.DBX7.0, 500 ms
   "2935RS001A01L01.DI.O_RANGE" : Bool AT %DB5075.DBX7.1, 500 ms
   "2935RS001A01L01.DI.SIG_FAULT" : Bool AT %DB5075.DBX7.2, 500 ms
   "2935RS001A01L01.DI.EnConfig" : Bool AT %DB5075.DBX7.3, 500 ms
   "2935RS001A01L01.DI.AEN" : Bool AT %DB5075.DBX7.4, 500 ms
   "2935RS001A01L01.DI.AL_SUPR" : Bool AT %DB5075.DBX7.5, 500 ms
   "2935RS001A01L01.Q.PV_NORM" : Real AT %DB5075.DBD8, 500 ms
   "2935RS001A01L01.Q.PV_SCAL" : Real AT %DB5075.DBD12, 500 ms
   "2935RS001A01L01.ParentInfo" : TextRef, internal   // Имя родителя для попап окна, вкладка инфо. При експорте из ECS через скрипт заполняется автоматически, если теги копируются в ручную то требуется в ручную задатать свойство Start Value

HMI tags "2935RS001A01L02"
   "2935RS001A01L02.MSW" : 52809b66-421d-457f-8884-6f7a49d4e247 AT %DB5076.DBX18.0, 500 ms
   "2935RS001A01L02.DefaultText" : TextRef, internal   // Заголовок POPUP окна. При експорте из ECS через скрипт заполняется автоматически, если теги копируются в ручную то требуется в ручную задатать свойство Start Value
   "2935RS001A01L02.BlockInfo" : Array [0..2] of Int AT %DB5076.DBX38.0, 500 ms
   "2935RS001A01L02.StatusWork" : Int AT %DB5076.DBW242, 500 ms
   "2935RS001A01L02.FP_PARAM.DampingTime" : Int AT %DB5076.DBW50, 500 ms
   "2935RS001A01L02.FP_PARAM.Force_Value" : Real AT %DB5076.DBD52, 500 ms
   "2935RS001A01L02.FP_PARAM.Scale_Min" : Real AT %DB5076.DBD56, 500 ms
   "2935RS001A01L02.FP_PARAM.Scale_Max" : Real AT %DB5076.DBD60, 500 ms
   "2935RS001A01L02.FP_PARAM.Gradient" : Real AT %DB5076.DBD64, 500 ms
   "2935RS001A01L02.FP_PARAM.Grad_Pos" : Real AT %DB5076.DBD68, 500 ms
   "2935RS001A01L02.FP_PARAM.Grad_Neg" : Real AT %DB5076.DBD72, 500 ms
   "2935RS001A01L02.FP_PARAM.Grad_X" : Real AT %DB5076.DBD76, 500 ms
   "2935RS001A01L02.FP_PARAM.Gradient_Time_Pre" : Int AT %DB5076.DBW80, 500 ms
   "2935RS001A01L02.FP_PARAM.Gradient_Time_ACC" : Int AT %DB5076.DBW82, 500 ms
   "2935RS001A01L02.FP_PARAM.Alarm_Hyst" : Real AT %DB5076.DBD84, 500 ms
   "2935RS001A01L02.FP_PARAM.AlarmLimit_H3" : Real AT %DB5076.DBD88, 500 ms
   "2935RS001A01L02.FP_PARAM.AlarmLimit_H2" : Real AT %DB5076.DBD92, 500 ms
   "2935RS001A01L02.FP_PARAM.AlarmLimit_H1" : Real AT %DB5076.DBD96, 500 ms
   "2935RS001A01L02.FP_PARAM.AlarmLimit_L1" : Real AT %DB5076.DBD100, 500 ms
   "2935RS001A01L02.FP_PARAM.AlarmLimit_L2" : Real AT %DB5076.DBD104, 500 ms
   "2935RS001A01L02.FP_PARAM.AlarmLimit_L3" : Real AT %DB5076.DBD108, 500 ms
   "2935RS001A01L02.FP_PARAM.AlarmDelay_H3_Pre" : Int AT %DB5076.DBW112, 500 ms
   "2935RS001A01L02.FP_PARAM.AlarmDelay_H3_Acc" : Int AT %DB5076.DBW114, 500 ms
   "2935RS001A01L02.FP_PARAM.AlarmDelay_H2_Pre" : Int AT %DB5076.DBW116, 500 ms
   "2935RS001A01L02.FP_PARAM.AlarmDelay_H2_Acc" : Int AT %DB5076.DBW118, 500 ms
   "2935RS001A01L02.FP_PARAM.AlarmDelay_H1_Pre" : Int AT %DB5076.DBW120, 500 ms
   "2935RS001A01L02.FP_PARAM.AlarmDelay_H1_Acc" : Int AT %DB5076.DBW122, 500 ms
   "2935RS001A01L02.FP_PARAM.AlarmDelay_L1_Pre" : Int AT %DB5076.DBW124, 500 ms
   "2935RS001A01L02.FP_PARAM.AlarmDelay_L1_Acc" : Int AT %DB5076.DBW126, 500 ms
   "2935RS001A01L02.FP_PARAM.AlarmDelay_L2_Pre" : Int AT %DB5076.DBW128, 500 ms
   "2935RS001A01L02.FP_PARAM.AlarmDelay_L2_Acc" : Int AT %DB5076.DBW130, 500 ms
   "2935RS001A01L02.FP_PARAM.AlarmDelay_L3_Pre" : Int AT %DB5076.DBW132, 500 ms
   "2935RS001A01L02.FP_PARAM.AlarmDelay_L3_Acc" : Int AT %DB5076.DBW134, 500 ms
   "2935RS001A01L02.FP_PARAM.OpenLoopDelay_Pre" : Int AT %DB5076.DBW136, 500 ms
   "2935RS001A01L02.FP_PARAM.OpenLoopDelay_Acc" : Int AT %DB5076.DBW138, 500 ms
   "2935RS001A01L02.FP_PARAM.OverRangeDelay_Pre" : Int AT %DB5076.DBW140, 500 ms
   "2935RS001A01L02.FP_PARAM.OverRangeDelay_Acc" : Int AT %DB5076.DBW142, 500 ms
   "2935RS001A01L02.FP_PARAM.AuxLimit_H2_Value" : Real AT %DB5076.DBD144, 500 ms
   "2935RS001A01L02.FP_PARAM.AuxLimit_H1_Value" : Real AT %DB5076.DBD148, 500 ms
   "2935RS001A01L02.FP_PARAM.AuxLimit_L2_Value" : Real AT %DB5076.DBD152, 500 ms
   "2935RS001A01L02.FP_PARAM.AuxLimit_L1_Value" : Real AT %DB5076.DBD156, 500 ms
   "2935RS001A01L02.Unit" : TextRef, internal   // Еденицы измерения При експорте из ECS через скрипт заполняется автоматически, если теги копируются в ручную то требуется задатать свойство Text
   "2935RS001A01L02.Decimals" : TextRef, internal   // Формат отображения При експорте из ECS через скрипт, заполняется автоматически. Если теги копируются в ручную то требуется задатать свойство Text s999999.9
   "2935RS001A01L02.FP_EN.Square" : Bool AT %DB5076.DBX46.0, 500 ms
   "2935RS001A01L02.FP_EN.SquareRoot" : Bool AT %DB5076.DBX46.1, 500 ms
   "2935RS001A01L02.FP_EN.ParentSupress" : Bool AT %DB5076.DBX46.2, 500 ms
   "2935RS001A01L02.FP_EN.ParentSupressUnit" : Bool AT %DB5076.DBX46.3, 500 ms
   "2935RS001A01L02.FP_EN.Force" : Bool AT %DB5076.DBX46.4, 500 ms
   "2935RS001A01L02.FP_EN.Damping" : Bool AT %DB5076.DBX46.5, 500 ms
   "2935RS001A01L02.FP_EN.Gradient_Pos" : Bool AT %DB5076.DBX46.6, 500 ms
   "2935RS001A01L02.FP_EN.Gradient_Neg" : Bool AT %DB5076.DBX46.7, 500 ms
   "2935RS001A01L02.FP_EN.Hysteresis" : Bool AT %DB5076.DBX47.0, 500 ms
   "2935RS001A01L02.FP_EN.Alarm_H3" : Bool AT %DB5076.DBX47.1, 500 ms
   "2935RS001A01L02.FP_EN.Alarm_H2" : Bool AT %DB5076.DBX47.2, 500 ms
   "2935RS001A01L02.FP_EN.Alarm_H1" : Bool AT %DB5076.DBX47.3, 500 ms
   "2935RS001A01L02.FP_EN.Alarm_L1" : Bool AT %DB5076.DBX47.4, 500 ms
   "2935RS001A01L02.FP_EN.Alarm_L2" : Bool AT %DB5076.DBX47.5, 500 ms
   "2935RS001A01L02.FP_EN.Alarm_L3" : Bool AT %DB5076.DBX47.6, 500 ms
   "2935RS001A01L02.FP_EN.AlarmDelay_H3" : Bool AT %DB5076.DBX47.7, 500 ms
   "2935RS001A01L02.FP_EN.AlarmDelay_H2" : Bool AT %DB5076.DBX48.0, 500 ms
   "2935RS001A01L02.FP_EN.AlarmDelay_H1" : Bool AT %DB5076.DBX48.1, 500 ms
   "2935RS001A01L02.FP_EN.AlarmDelay_L1" : Bool AT %DB5076.DBX48.2, 500 ms
   "2935RS001A01L02.FP_EN.AlarmDelay_L2" : Bool AT %DB5076.DBX48.3, 500 ms
   "2935RS001A01L02.FP_EN.AlarmDelay_L3" : Bool AT %DB5076.DBX48.4, 500 ms
   "2935RS001A01L02.FP_EN.ROC_Warn" : Bool AT %DB5076.DBX48.5, 500 ms
   "2935RS001A01L02.FP_EN.U_Range_Warn" : Bool AT %DB5076.DBX48.6, 500 ms
   "2935RS001A01L02.FP_EN.O_Range_Warn" : Bool AT %DB5076.DBX48.7, 500 ms
   "2935RS001A01L02.trend_tag_name" : TextRef, internal   // Еденицы измерения При експорте из ECS через скрипт - заполняется автоматически, если теги копируются в ручную то требуется задатать свойство Text - имя тега для тренда
   "2935RS001A01L02.DQ.AL_H3" : Bool AT %DB5076.DBX16.0, 500 ms
   "2935RS001A01L02.DQ.AL_H2" : Bool AT %DB5076.DBX16.1, 500 ms
   "2935RS001A01L02.DQ.AL_H1" : Bool AT %DB5076.DBX16.2, 500 ms
   "2935RS001A01L02.DQ.AL_L1" : Bool AT %DB5076.DBX16.3, 500 ms
   "2935RS001A01L02.DQ.AL_L2" : Bool AT %DB5076.DBX16.4, 500 ms
   "2935RS001A01L02.DQ.AL_L3" : Bool AT %DB5076.DBX16.5, 500 ms
   "2935RS001A01L02.DQ.SIG_OK" : Bool AT %DB5076.DBX16.6, 500 ms
   "2935RS001A01L02.DQ.LIM_H2" : Bool AT %DB5076.DBX16.7, 500 ms
   "2935RS001A01L02.DQ.LIM_H1" : Bool AT %DB5076.DBX17.0, 500 ms
   "2935RS001A01L02.DQ.LIM_L1" : Bool AT %DB5076.DBX17.1, 500 ms
   "2935RS001A01L02.DQ.LIM_L2" : Bool AT %DB5076.DBX17.2, 500 ms
   "2935RS001A01L02.DQ.GR_P" : Bool AT %DB5076.DBX17.3, 500 ms
   "2935RS001A01L02.DQ.GR_N" : Bool AT %DB5076.DBX17.4, 500 ms
   "2935RS001A01L02.I.IN" : Real AT %DB5076.DBD2, 500 ms
   "2935RS001A01L02.I.SIG_TYPE" : Int AT %DB5076.DBW0, 500 ms
   "2935RS001A01L02.I.FI_BUS" : Byte AT %DB5076.DBB6, 500 ms
   "2935RS001A01L02.DI.U_RANGE" : Bool AT %DB5076.DBX7.0, 500 ms
   "2935RS001A01L02.DI.O_RANGE" : Bool AT %DB5076.DBX7.1, 500 ms
   "2935RS001A01L02.DI.SIG_FAULT" : Bool AT %DB5076.DBX7.2, 500 ms
   "2935RS001A01L02.DI.EnConfig" : Bool AT %DB5076.DBX7.3, 500 ms
   "2935RS001A01L02.DI.AEN" : Bool AT %DB5076.DBX7.4, 500 ms
   "2935RS001A01L02.DI.AL_SUPR" : Bool AT %DB5076.DBX7.5, 500 ms
   "2935RS001A01L02.Q.PV_NORM" : Real AT %DB5076.DBD8, 500 ms
   "2935RS001A01L02.Q.PV_SCAL" : Real AT %DB5076.DBD12, 500 ms
   "2935RS001A01L02.ParentInfo" : TextRef, internal   // Имя родителя для попап окна, вкладка инфо. При експорте из ECS через скрипт заполняется автоматически, если теги копируются в ручную то требуется в ручную задатать свойство Start Value

HMI tags "2935RS001A01T01"
   "2935RS001A01T01.MSW" : 52809b66-421d-457f-8884-6f7a49d4e247 AT %DB5077.DBX18.0, 500 ms
   "2935RS001A01T01.DefaultText" : TextRef, internal   // Заголовок POPUP окна. При експорте из ECS через скрипт заполняется автоматически, если теги копируются в ручную то требуется в ручную задатать свойство Start Value
   "2935RS001A01T01.BlockInfo" : Array [0..2] of Int AT %DB5077.DBX38.0, 500 ms
   "2935RS001A01T01.StatusWork" : Int AT %DB5077.DBW242, 500 ms
   "2935RS001A01T01.FP_PARAM.DampingTime" : Int AT %DB5077.DBW50, 500 ms
   "2935RS001A01T01.FP_PARAM.Force_Value" : Real AT %DB5077.DBD52, 500 ms
   "2935RS001A01T01.FP_PARAM.Scale_Min" : Real AT %DB5077.DBD56, 500 ms
   "2935RS001A01T01.FP_PARAM.Scale_Max" : Real AT %DB5077.DBD60, 500 ms
   "2935RS001A01T01.FP_PARAM.Gradient" : Real AT %DB5077.DBD64, 500 ms
   "2935RS001A01T01.FP_PARAM.Grad_Pos" : Real AT %DB5077.DBD68, 500 ms
   "2935RS001A01T01.FP_PARAM.Grad_Neg" : Real AT %DB5077.DBD72, 500 ms
   "2935RS001A01T01.FP_PARAM.Grad_X" : Real AT %DB5077.DBD76, 500 ms
   "2935RS001A01T01.FP_PARAM.Gradient_Time_Pre" : Int AT %DB5077.DBW80, 500 ms
   "2935RS001A01T01.FP_PARAM.Gradient_Time_ACC" : Int AT %DB5077.DBW82, 500 ms
   "2935RS001A01T01.FP_PARAM.Alarm_Hyst" : Real AT %DB5077.DBD84, 500 ms
   "2935RS001A01T01.FP_PARAM.AlarmLimit_H3" : Real AT %DB5077.DBD88, 500 ms
   "2935RS001A01T01.FP_PARAM.AlarmLimit_H2" : Real AT %DB5077.DBD92, 500 ms
   "2935RS001A01T01.FP_PARAM.AlarmLimit_H1" : Real AT %DB5077.DBD96, 500 ms
   "2935RS001A01T01.FP_PARAM.AlarmLimit_L1" : Real AT %DB5077.DBD100, 500 ms
   "2935RS001A01T01.FP_PARAM.AlarmLimit_L2" : Real AT %DB5077.DBD104, 500 ms
   "2935RS001A01T01.FP_PARAM.AlarmLimit_L3" : Real AT %DB5077.DBD108, 500 ms
   "2935RS001A01T01.FP_PARAM.AlarmDelay_H3_Pre" : Int AT %DB5077.DBW112, 500 ms
   "2935RS001A01T01.FP_PARAM.AlarmDelay_H3_Acc" : Int AT %DB5077.DBW114, 500 ms
   "2935RS001A01T01.FP_PARAM.AlarmDelay_H2_Pre" : Int AT %DB5077.DBW116, 500 ms
   "2935RS001A01T01.FP_PARAM.AlarmDelay_H2_Acc" : Int AT %DB5077.DBW118, 500 ms
   "2935RS001A01T01.FP_PARAM.AlarmDelay_H1_Pre" : Int AT %DB5077.DBW120, 500 ms
   "2935RS001A01T01.FP_PARAM.AlarmDelay_H1_Acc" : Int AT %DB5077.DBW122, 500 ms
   "2935RS001A01T01.FP_PARAM.AlarmDelay_L1_Pre" : Int AT %DB5077.DBW124, 500 ms
   "2935RS001A01T01.FP_PARAM.AlarmDelay_L1_Acc" : Int AT %DB5077.DBW126, 500 ms
   "2935RS001A01T01.FP_PARAM.AlarmDelay_L2_Pre" : Int AT %DB5077.DBW128, 500 ms
   "2935RS001A01T01.FP_PARAM.AlarmDelay_L2_Acc" : Int AT %DB5077.DBW130, 500 ms
   "2935RS001A01T01.FP_PARAM.AlarmDelay_L3_Pre" : Int AT %DB5077.DBW132, 500 ms
   "2935RS001A01T01.FP_PARAM.AlarmDelay_L3_Acc" : Int AT %DB5077.DBW134, 500 ms
   "2935RS001A01T01.FP_PARAM.OpenLoopDelay_Pre" : Int AT %DB5077.DBW136, 500 ms
   "2935RS001A01T01.FP_PARAM.OpenLoopDelay_Acc" : Int AT %DB5077.DBW138, 500 ms
   "2935RS001A01T01.FP_PARAM.OverRangeDelay_Pre" : Int AT %DB5077.DBW140, 500 ms
   "2935RS001A01T01.FP_PARAM.OverRangeDelay_Acc" : Int AT %DB5077.DBW142, 500 ms
   "2935RS001A01T01.FP_PARAM.AuxLimit_H2_Value" : Real AT %DB5077.DBD144, 500 ms
   "2935RS001A01T01.FP_PARAM.AuxLimit_H1_Value" : Real AT %DB5077.DBD148, 500 ms
   "2935RS001A01T01.FP_PARAM.AuxLimit_L2_Value" : Real AT %DB5077.DBD152, 500 ms
   "2935RS001A01T01.FP_PARAM.AuxLimit_L1_Value" : Real AT %DB5077.DBD156, 500 ms
   "2935RS001A01T01.Unit" : TextRef, internal   // Еденицы измерения При експорте из ECS через скрипт заполняется автоматически, если теги копируются в ручную то требуется задатать свойство Text
   "2935RS001A01T01.Decimals" : TextRef, internal   // Формат отображения При експорте из ECS через скрипт, заполняется автоматически. Если теги копируются в ручную то требуется задатать свойство Text s999999.9
   "2935RS001A01T01.FP_EN.Square" : Bool AT %DB5077.DBX46.0, 500 ms
   "2935RS001A01T01.FP_EN.SquareRoot" : Bool AT %DB5077.DBX46.1, 500 ms
   "2935RS001A01T01.FP_EN.ParentSupress" : Bool AT %DB5077.DBX46.2, 500 ms
   "2935RS001A01T01.FP_EN.ParentSupressUnit" : Bool AT %DB5077.DBX46.3, 500 ms
   "2935RS001A01T01.FP_EN.Force" : Bool AT %DB5077.DBX46.4, 500 ms
   "2935RS001A01T01.FP_EN.Damping" : Bool AT %DB5077.DBX46.5, 500 ms
   "2935RS001A01T01.FP_EN.Gradient_Pos" : Bool AT %DB5077.DBX46.6, 500 ms
   "2935RS001A01T01.FP_EN.Gradient_Neg" : Bool AT %DB5077.DBX46.7, 500 ms
   "2935RS001A01T01.FP_EN.Hysteresis" : Bool AT %DB5077.DBX47.0, 500 ms
   "2935RS001A01T01.FP_EN.Alarm_H3" : Bool AT %DB5077.DBX47.1, 500 ms
   "2935RS001A01T01.FP_EN.Alarm_H2" : Bool AT %DB5077.DBX47.2, 500 ms
   "2935RS001A01T01.FP_EN.Alarm_H1" : Bool AT %DB5077.DBX47.3, 500 ms
   "2935RS001A01T01.FP_EN.Alarm_L1" : Bool AT %DB5077.DBX47.4, 500 ms
   "2935RS001A01T01.FP_EN.Alarm_L2" : Bool AT %DB5077.DBX47.5, 500 ms
   "2935RS001A01T01.FP_EN.Alarm_L3" : Bool AT %DB5077.DBX47.6, 500 ms
   "2935RS001A01T01.FP_EN.AlarmDelay_H3" : Bool AT %DB5077.DBX47.7, 500 ms
   "2935RS001A01T01.FP_EN.AlarmDelay_H2" : Bool AT %DB5077.DBX48.0, 500 ms
   "2935RS001A01T01.FP_EN.AlarmDelay_H1" : Bool AT %DB5077.DBX48.1, 500 ms
   "2935RS001A01T01.FP_EN.AlarmDelay_L1" : Bool AT %DB5077.DBX48.2, 500 ms
   "2935RS001A01T01.FP_EN.AlarmDelay_L2" : Bool AT %DB5077.DBX48.3, 500 ms
   "2935RS001A01T01.FP_EN.AlarmDelay_L3" : Bool AT %DB5077.DBX48.4, 500 ms
   "2935RS001A01T01.FP_EN.ROC_Warn" : Bool AT %DB5077.DBX48.5, 500 ms
   "2935RS001A01T01.FP_EN.U_Range_Warn" : Bool AT %DB5077.DBX48.6, 500 ms
   "2935RS001A01T01.FP_EN.O_Range_Warn" : Bool AT %DB5077.DBX48.7, 500 ms
   "2935RS001A01T01.trend_tag_name" : TextRef, internal   // Еденицы измерения При експорте из ECS через скрипт - заполняется автоматически, если теги копируются в ручную то требуется задатать свойство Text - имя тега для тренда
   "2935RS001A01T01.DQ.AL_H3" : Bool AT %DB5077.DBX16.0, 500 ms
   "2935RS001A01T01.DQ.AL_H2" : Bool AT %DB5077.DBX16.1, 500 ms
   "2935RS001A01T01.DQ.AL_H1" : Bool AT %DB5077.DBX16.2, 500 ms
   "2935RS001A01T01.DQ.AL_L1" : Bool AT %DB5077.DBX16.3, 500 ms
   "2935RS001A01T01.DQ.AL_L2" : Bool AT %DB5077.DBX16.4, 500 ms
   "2935RS001A01T01.DQ.AL_L3" : Bool AT %DB5077.DBX16.5, 500 ms
   "2935RS001A01T01.DQ.SIG_OK" : Bool AT %DB5077.DBX16.6, 500 ms
   "2935RS001A01T01.DQ.LIM_H2" : Bool AT %DB5077.DBX16.7, 500 ms
   "2935RS001A01T01.DQ.LIM_H1" : Bool AT %DB5077.DBX17.0, 500 ms
   "2935RS001A01T01.DQ.LIM_L1" : Bool AT %DB5077.DBX17.1, 500 ms
   "2935RS001A01T01.DQ.LIM_L2" : Bool AT %DB5077.DBX17.2, 500 ms
   "2935RS001A01T01.DQ.GR_P" : Bool AT %DB5077.DBX17.3, 500 ms
   "2935RS001A01T01.DQ.GR_N" : Bool AT %DB5077.DBX17.4, 500 ms
   "2935RS001A01T01.I.IN" : Real AT %DB5077.DBD2, 500 ms
   "2935RS001A01T01.I.SIG_TYPE" : Int AT %DB5077.DBW0, 500 ms
   "2935RS001A01T01.I.FI_BUS" : Byte AT %DB5077.DBB6, 500 ms
   "2935RS001A01T01.DI.U_RANGE" : Bool AT %DB5077.DBX7.0, 500 ms
   "2935RS001A01T01.DI.O_RANGE" : Bool AT %DB5077.DBX7.1, 500 ms
   "2935RS001A01T01.DI.SIG_FAULT" : Bool AT %DB5077.DBX7.2, 500 ms
   "2935RS001A01T01.DI.EnConfig" : Bool AT %DB5077.DBX7.3, 500 ms
   "2935RS001A01T01.DI.AEN" : Bool AT %DB5077.DBX7.4, 500 ms
   "2935RS001A01T01.DI.AL_SUPR" : Bool AT %DB5077.DBX7.5, 500 ms
   "2935RS001A01T01.Q.PV_NORM" : Real AT %DB5077.DBD8, 500 ms
   "2935RS001A01T01.Q.PV_SCAL" : Real AT %DB5077.DBD12, 500 ms
   "2935RS001A01T01.ParentInfo" : TextRef, internal   // Имя родителя для попап окна, вкладка инфо. При експорте из ECS через скрипт заполняется автоматически, если теги копируются в ручную то требуется в ручную задатать свойство Start Value

HMI tags "2935RS001A01T02"
   "2935RS001A01T02.MSW" : 52809b66-421d-457f-8884-6f7a49d4e247 AT %DB5078.DBX18.0, 500 ms
   "2935RS001A01T02.DefaultText" : TextRef, internal   // Заголовок POPUP окна. При експорте из ECS через скрипт заполняется автоматически, если теги копируются в ручную то требуется в ручную задатать свойство Start Value
   "2935RS001A01T02.BlockInfo" : Array [0..2] of Int AT %DB5078.DBX38.0, 500 ms
   "2935RS001A01T02.StatusWork" : Int AT %DB5078.DBW242, 500 ms
   "2935RS001A01T02.FP_PARAM.DampingTime" : Int AT %DB5078.DBW50, 500 ms
   "2935RS001A01T02.FP_PARAM.Force_Value" : Real AT %DB5078.DBD52, 500 ms
   "2935RS001A01T02.FP_PARAM.Scale_Min" : Real AT %DB5078.DBD56, 500 ms
   "2935RS001A01T02.FP_PARAM.Scale_Max" : Real AT %DB5078.DBD60, 500 ms
   "2935RS001A01T02.FP_PARAM.Gradient" : Real AT %DB5078.DBD64, 500 ms
   "2935RS001A01T02.FP_PARAM.Grad_Pos" : Real AT %DB5078.DBD68, 500 ms
   "2935RS001A01T02.FP_PARAM.Grad_Neg" : Real AT %DB5078.DBD72, 500 ms
   "2935RS001A01T02.FP_PARAM.Grad_X" : Real AT %DB5078.DBD76, 500 ms
   "2935RS001A01T02.FP_PARAM.Gradient_Time_Pre" : Int AT %DB5078.DBW80, 500 ms
   "2935RS001A01T02.FP_PARAM.Gradient_Time_ACC" : Int AT %DB5078.DBW82, 500 ms
   "2935RS001A01T02.FP_PARAM.Alarm_Hyst" : Real AT %DB5078.DBD84, 500 ms
   "2935RS001A01T02.FP_PARAM.AlarmLimit_H3" : Real AT %DB5078.DBD88, 500 ms
   "2935RS001A01T02.FP_PARAM.AlarmLimit_H2" : Real AT %DB5078.DBD92, 500 ms
   "2935RS001A01T02.FP_PARAM.AlarmLimit_H1" : Real AT %DB5078.DBD96, 500 ms
   "2935RS001A01T02.FP_PARAM.AlarmLimit_L1" : Real AT %DB5078.DBD100, 500 ms
   "2935RS001A01T02.FP_PARAM.AlarmLimit_L2" : Real AT %DB5078.DBD104, 500 ms
   "2935RS001A01T02.FP_PARAM.AlarmLimit_L3" : Real AT %DB5078.DBD108, 500 ms
   "2935RS001A01T02.FP_PARAM.AlarmDelay_H3_Pre" : Int AT %DB5078.DBW112, 500 ms
   "2935RS001A01T02.FP_PARAM.AlarmDelay_H3_Acc" : Int AT %DB5078.DBW114, 500 ms
   "2935RS001A01T02.FP_PARAM.AlarmDelay_H2_Pre" : Int AT %DB5078.DBW116, 500 ms
   "2935RS001A01T02.FP_PARAM.AlarmDelay_H2_Acc" : Int AT %DB5078.DBW118, 500 ms
   "2935RS001A01T02.FP_PARAM.AlarmDelay_H1_Pre" : Int AT %DB5078.DBW120, 500 ms
   "2935RS001A01T02.FP_PARAM.AlarmDelay_H1_Acc" : Int AT %DB5078.DBW122, 500 ms
   "2935RS001A01T02.FP_PARAM.AlarmDelay_L1_Pre" : Int AT %DB5078.DBW124, 500 ms
   "2935RS001A01T02.FP_PARAM.AlarmDelay_L1_Acc" : Int AT %DB5078.DBW126, 500 ms
   "2935RS001A01T02.FP_PARAM.AlarmDelay_L2_Pre" : Int AT %DB5078.DBW128, 500 ms
   "2935RS001A01T02.FP_PARAM.AlarmDelay_L2_Acc" : Int AT %DB5078.DBW130, 500 ms
   "2935RS001A01T02.FP_PARAM.AlarmDelay_L3_Pre" : Int AT %DB5078.DBW132, 500 ms
   "2935RS001A01T02.FP_PARAM.AlarmDelay_L3_Acc" : Int AT %DB5078.DBW134, 500 ms
   "2935RS001A01T02.FP_PARAM.OpenLoopDelay_Pre" : Int AT %DB5078.DBW136, 500 ms
   "2935RS001A01T02.FP_PARAM.OpenLoopDelay_Acc" : Int AT %DB5078.DBW138, 500 ms
   "2935RS001A01T02.FP_PARAM.OverRangeDelay_Pre" : Int AT %DB5078.DBW140, 500 ms
   "2935RS001A01T02.FP_PARAM.OverRangeDelay_Acc" : Int AT %DB5078.DBW142, 500 ms
   "2935RS001A01T02.FP_PARAM.AuxLimit_H2_Value" : Real AT %DB5078.DBD144, 500 ms
   "2935RS001A01T02.FP_PARAM.AuxLimit_H1_Value" : Real AT %DB5078.DBD148, 500 ms
   "2935RS001A01T02.FP_PARAM.AuxLimit_L2_Value" : Real AT %DB5078.DBD152, 500 ms
   "2935RS001A01T02.FP_PARAM.AuxLimit_L1_Value" : Real AT %DB5078.DBD156, 500 ms
   "2935RS001A01T02.Unit" : TextRef, internal   // Еденицы измерения При експорте из ECS через скрипт заполняется автоматически, если теги копируются в ручную то требуется задатать свойство Text
   "2935RS001A01T02.Decimals" : TextRef, internal   // Формат отображения При експорте из ECS через скрипт, заполняется автоматически. Если теги копируются в ручную то требуется задатать свойство Text s999999.9
   "2935RS001A01T02.FP_EN.Square" : Bool AT %DB5078.DBX46.0, 500 ms
   "2935RS001A01T02.FP_EN.SquareRoot" : Bool AT %DB5078.DBX46.1, 500 ms
   "2935RS001A01T02.FP_EN.ParentSupress" : Bool AT %DB5078.DBX46.2, 500 ms
   "2935RS001A01T02.FP_EN.ParentSupressUnit" : Bool AT %DB5078.DBX46.3, 500 ms
   "2935RS001A01T02.FP_EN.Force" : Bool AT %DB5078.DBX46.4, 500 ms
   "2935RS001A01T02.FP_EN.Damping" : Bool AT %DB5078.DBX46.5, 500 ms
   "2935RS001A01T02.FP_EN.Gradient_Pos" : Bool AT %DB5078.DBX46.6, 500 ms
   "2935RS001A01T02.FP_EN.Gradient_Neg" : Bool AT %DB5078.DBX46.7, 500 ms
   "2935RS001A01T02.FP_EN.Hysteresis" : Bool AT %DB5078.DBX47.0, 500 ms
   "2935RS001A01T02.FP_EN.Alarm_H3" : Bool AT %DB5078.DBX47.1, 500 ms
   "2935RS001A01T02.FP_EN.Alarm_H2" : Bool AT %DB5078.DBX47.2, 500 ms
   "2935RS001A01T02.FP_EN.Alarm_H1" : Bool AT %DB5078.DBX47.3, 500 ms
   "2935RS001A01T02.FP_EN.Alarm_L1" : Bool AT %DB5078.DBX47.4, 500 ms
   "2935RS001A01T02.FP_EN.Alarm_L2" : Bool AT %DB5078.DBX47.5, 500 ms
   "2935RS001A01T02.FP_EN.Alarm_L3" : Bool AT %DB5078.DBX47.6, 500 ms
   "2935RS001A01T02.FP_EN.AlarmDelay_H3" : Bool AT %DB5078.DBX47.7, 500 ms
   "2935RS001A01T02.FP_EN.AlarmDelay_H2" : Bool AT %DB5078.DBX48.0, 500 ms
   "2935RS001A01T02.FP_EN.AlarmDelay_H1" : Bool AT %DB5078.DBX48.1, 500 ms
   "2935RS001A01T02.FP_EN.AlarmDelay_L1" : Bool AT %DB5078.DBX48.2, 500 ms
   "2935RS001A01T02.FP_EN.AlarmDelay_L2" : Bool AT %DB5078.DBX48.3, 500 ms
   "2935RS001A01T02.FP_EN.AlarmDelay_L3" : Bool AT %DB5078.DBX48.4, 500 ms
   "2935RS001A01T02.FP_EN.ROC_Warn" : Bool AT %DB5078.DBX48.5, 500 ms
   "2935RS001A01T02.FP_EN.U_Range_Warn" : Bool AT %DB5078.DBX48.6, 500 ms
   "2935RS001A01T02.FP_EN.O_Range_Warn" : Bool AT %DB5078.DBX48.7, 500 ms
   "2935RS001A01T02.trend_tag_name" : TextRef, internal   // Еденицы измерения При експорте из ECS через скрипт - заполняется автоматически, если теги копируются в ручную то требуется задатать свойство Text - имя тега для тренда
   "2935RS001A01T02.DQ.AL_H3" : Bool AT %DB5078.DBX16.0, 500 ms
   "2935RS001A01T02.DQ.AL_H2" : Bool AT %DB5078.DBX16.1, 500 ms
   "2935RS001A01T02.DQ.AL_H1" : Bool AT %DB5078.DBX16.2, 500 ms
   "2935RS001A01T02.DQ.AL_L1" : Bool AT %DB5078.DBX16.3, 500 ms
   "2935RS001A01T02.DQ.AL_L2" : Bool AT %DB5078.DBX16.4, 500 ms
   "2935RS001A01T02.DQ.AL_L3" : Bool AT %DB5078.DBX16.5, 500 ms
   "2935RS001A01T02.DQ.SIG_OK" : Bool AT %DB5078.DBX16.6, 500 ms
   "2935RS001A01T02.DQ.LIM_H2" : Bool AT %DB5078.DBX16.7, 500 ms
   "2935RS001A01T02.DQ.LIM_H1" : Bool AT %DB5078.DBX17.0, 500 ms
   "2935RS001A01T02.DQ.LIM_L1" : Bool AT %DB5078.DBX17.1, 500 ms
   "2935RS001A01T02.DQ.LIM_L2" : Bool AT %DB5078.DBX17.2, 500 ms
   "2935RS001A01T02.DQ.GR_P" : Bool AT %DB5078.DBX17.3, 500 ms
   "2935RS001A01T02.DQ.GR_N" : Bool AT %DB5078.DBX17.4, 500 ms
   "2935RS001A01T02.I.IN" : Real AT %DB5078.DBD2, 500 ms
   "2935RS001A01T02.I.SIG_TYPE" : Int AT %DB5078.DBW0, 500 ms
   "2935RS001A01T02.I.FI_BUS" : Byte AT %DB5078.DBB6, 500 ms
   "2935RS001A01T02.DI.U_RANGE" : Bool AT %DB5078.DBX7.0, 500 ms
   "2935RS001A01T02.DI.O_RANGE" : Bool AT %DB5078.DBX7.1, 500 ms
   "2935RS001A01T02.DI.SIG_FAULT" : Bool AT %DB5078.DBX7.2, 500 ms
   "2935RS001A01T02.DI.EnConfig" : Bool AT %DB5078.DBX7.3, 500 ms
   "2935RS001A01T02.DI.AEN" : Bool AT %DB5078.DBX7.4, 500 ms
   "2935RS001A01T02.DI.AL_SUPR" : Bool AT %DB5078.DBX7.5, 500 ms
   "2935RS001A01T02.Q.PV_NORM" : Real AT %DB5078.DBD8, 500 ms
   "2935RS001A01T02.Q.PV_SCAL" : Real AT %DB5078.DBD12, 500 ms
   "2935RS001A01T02.ParentInfo" : TextRef, internal   // Имя родителя для попап окна, вкладка инфо. При експорте из ECS через скрипт заполняется автоматически, если теги копируются в ручную то требуется в ручную задатать свойство Start Value

HMI tags "2935RS001A01T03"
   "2935RS001A01T03.MSW" : 52809b66-421d-457f-8884-6f7a49d4e247 AT %DB5079.DBX18.0, 500 ms
   "2935RS001A01T03.DefaultText" : TextRef, internal   // Заголовок POPUP окна. При експорте из ECS через скрипт заполняется автоматически, если теги копируются в ручную то требуется в ручную задатать свойство Start Value
   "2935RS001A01T03.BlockInfo" : Array [0..2] of Int AT %DB5079.DBX38.0, 500 ms
   "2935RS001A01T03.StatusWork" : Int AT %DB5079.DBW242, 500 ms
   "2935RS001A01T03.FP_PARAM.DampingTime" : Int AT %DB5079.DBW50, 500 ms
   "2935RS001A01T03.FP_PARAM.Force_Value" : Real AT %DB5079.DBD52, 500 ms
   "2935RS001A01T03.FP_PARAM.Scale_Min" : Real AT %DB5079.DBD56, 500 ms
   "2935RS001A01T03.FP_PARAM.Scale_Max" : Real AT %DB5079.DBD60, 500 ms
   "2935RS001A01T03.FP_PARAM.Gradient" : Real AT %DB5079.DBD64, 500 ms
   "2935RS001A01T03.FP_PARAM.Grad_Pos" : Real AT %DB5079.DBD68, 500 ms
   "2935RS001A01T03.FP_PARAM.Grad_Neg" : Real AT %DB5079.DBD72, 500 ms
   "2935RS001A01T03.FP_PARAM.Grad_X" : Real AT %DB5079.DBD76, 500 ms
   "2935RS001A01T03.FP_PARAM.Gradient_Time_Pre" : Int AT %DB5079.DBW80, 500 ms
   "2935RS001A01T03.FP_PARAM.Gradient_Time_ACC" : Int AT %DB5079.DBW82, 500 ms
   "2935RS001A01T03.FP_PARAM.Alarm_Hyst" : Real AT %DB5079.DBD84, 500 ms
   "2935RS001A01T03.FP_PARAM.AlarmLimit_H3" : Real AT %DB5079.DBD88, 500 ms
   "2935RS001A01T03.FP_PARAM.AlarmLimit_H2" : Real AT %DB5079.DBD92, 500 ms
   "2935RS001A01T03.FP_PARAM.AlarmLimit_H1" : Real AT %DB5079.DBD96, 500 ms
   "2935RS001A01T03.FP_PARAM.AlarmLimit_L1" : Real AT %DB5079.DBD100, 500 ms
   "2935RS001A01T03.FP_PARAM.AlarmLimit_L2" : Real AT %DB5079.DBD104, 500 ms
   "2935RS001A01T03.FP_PARAM.AlarmLimit_L3" : Real AT %DB5079.DBD108, 500 ms
   "2935RS001A01T03.FP_PARAM.AlarmDelay_H3_Pre" : Int AT %DB5079.DBW112, 500 ms
   "2935RS001A01T03.FP_PARAM.AlarmDelay_H3_Acc" : Int AT %DB5079.DBW114, 500 ms
   "2935RS001A01T03.FP_PARAM.AlarmDelay_H2_Pre" : Int AT %DB5079.DBW116, 500 ms
   "2935RS001A01T03.FP_PARAM.AlarmDelay_H2_Acc" : Int AT %DB5079.DBW118, 500 ms
   "2935RS001A01T03.FP_PARAM.AlarmDelay_H1_Pre" : Int AT %DB5079.DBW120, 500 ms
   "2935RS001A01T03.FP_PARAM.AlarmDelay_H1_Acc" : Int AT %DB5079.DBW122, 500 ms
   "2935RS001A01T03.FP_PARAM.AlarmDelay_L1_Pre" : Int AT %DB5079.DBW124, 500 ms
   "2935RS001A01T03.FP_PARAM.AlarmDelay_L1_Acc" : Int AT %DB5079.DBW126, 500 ms
   "2935RS001A01T03.FP_PARAM.AlarmDelay_L2_Pre" : Int AT %DB5079.DBW128, 500 ms
   "2935RS001A01T03.FP_PARAM.AlarmDelay_L2_Acc" : Int AT %DB5079.DBW130, 500 ms
   "2935RS001A01T03.FP_PARAM.AlarmDelay_L3_Pre" : Int AT %DB5079.DBW132, 500 ms
   "2935RS001A01T03.FP_PARAM.AlarmDelay_L3_Acc" : Int AT %DB5079.DBW134, 500 ms
   "2935RS001A01T03.FP_PARAM.OpenLoopDelay_Pre" : Int AT %DB5079.DBW136, 500 ms
   "2935RS001A01T03.FP_PARAM.OpenLoopDelay_Acc" : Int AT %DB5079.DBW138, 500 ms
   "2935RS001A01T03.FP_PARAM.OverRangeDelay_Pre" : Int AT %DB5079.DBW140, 500 ms
   "2935RS001A01T03.FP_PARAM.OverRangeDelay_Acc" : Int AT %DB5079.DBW142, 500 ms
   "2935RS001A01T03.FP_PARAM.AuxLimit_H2_Value" : Real AT %DB5079.DBD144, 500 ms
   "2935RS001A01T03.FP_PARAM.AuxLimit_H1_Value" : Real AT %DB5079.DBD148, 500 ms
   "2935RS001A01T03.FP_PARAM.AuxLimit_L2_Value" : Real AT %DB5079.DBD152, 500 ms
   "2935RS001A01T03.FP_PARAM.AuxLimit_L1_Value" : Real AT %DB5079.DBD156, 500 ms
   "2935RS001A01T03.Unit" : TextRef, internal   // Еденицы измерения При експорте из ECS через скрипт заполняется автоматически, если теги копируются в ручную то требуется задатать свойство Text
   "2935RS001A01T03.Decimals" : TextRef, internal   // Формат отображения При експорте из ECS через скрипт, заполняется автоматически. Если теги копируются в ручную то требуется задатать свойство Text s999999.9
   "2935RS001A01T03.FP_EN.Square" : Bool AT %DB5079.DBX46.0, 500 ms
   "2935RS001A01T03.FP_EN.SquareRoot" : Bool AT %DB5079.DBX46.1, 500 ms
   "2935RS001A01T03.FP_EN.ParentSupress" : Bool AT %DB5079.DBX46.2, 500 ms
   "2935RS001A01T03.FP_EN.ParentSupressUnit" : Bool AT %DB5079.DBX46.3, 500 ms
   "2935RS001A01T03.FP_EN.Force" : Bool AT %DB5079.DBX46.4, 500 ms
   "2935RS001A01T03.FP_EN.Damping" : Bool AT %DB5079.DBX46.5, 500 ms
   "2935RS001A01T03.FP_EN.Gradient_Pos" : Bool AT %DB5079.DBX46.6, 500 ms
   "2935RS001A01T03.FP_EN.Gradient_Neg" : Bool AT %DB5079.DBX46.7, 500 ms
   "2935RS001A01T03.FP_EN.Hysteresis" : Bool AT %DB5079.DBX47.0, 500 ms
   "2935RS001A01T03.FP_EN.Alarm_H3" : Bool AT %DB5079.DBX47.1, 500 ms
   "2935RS001A01T03.FP_EN.Alarm_H2" : Bool AT %DB5079.DBX47.2, 500 ms
   "2935RS001A01T03.FP_EN.Alarm_H1" : Bool AT %DB5079.DBX47.3, 500 ms
   "2935RS001A01T03.FP_EN.Alarm_L1" : Bool AT %DB5079.DBX47.4, 500 ms
   "2935RS001A01T03.FP_EN.Alarm_L2" : Bool AT %DB5079.DBX47.5, 500 ms
   "2935RS001A01T03.FP_EN.Alarm_L3" : Bool AT %DB5079.DBX47.6, 500 ms
   "2935RS001A01T03.FP_EN.AlarmDelay_H3" : Bool AT %DB5079.DBX47.7, 500 ms
   "2935RS001A01T03.FP_EN.AlarmDelay_H2" : Bool AT %DB5079.DBX48.0, 500 ms
   "2935RS001A01T03.FP_EN.AlarmDelay_H1" : Bool AT %DB5079.DBX48.1, 500 ms
   "2935RS001A01T03.FP_EN.AlarmDelay_L1" : Bool AT %DB5079.DBX48.2, 500 ms
   "2935RS001A01T03.FP_EN.AlarmDelay_L2" : Bool AT %DB5079.DBX48.3, 500 ms
   "2935RS001A01T03.FP_EN.AlarmDelay_L3" : Bool AT %DB5079.DBX48.4, 500 ms
   "2935RS001A01T03.FP_EN.ROC_Warn" : Bool AT %DB5079.DBX48.5, 500 ms
   "2935RS001A01T03.FP_EN.U_Range_Warn" : Bool AT %DB5079.DBX48.6, 500 ms
   "2935RS001A01T03.FP_EN.O_Range_Warn" : Bool AT %DB5079.DBX48.7, 500 ms
   "2935RS001A01T03.trend_tag_name" : TextRef, internal   // Еденицы измерения При експорте из ECS через скрипт - заполняется автоматически, если теги копируются в ручную то требуется задатать свойство Text - имя тега для тренда
   "2935RS001A01T03.DQ.AL_H3" : Bool AT %DB5079.DBX16.0, 500 ms
   "2935RS001A01T03.DQ.AL_H2" : Bool AT %DB5079.DBX16.1, 500 ms
   "2935RS001A01T03.DQ.AL_H1" : Bool AT %DB5079.DBX16.2, 500 ms
   "2935RS001A01T03.DQ.AL_L1" : Bool AT %DB5079.DBX16.3, 500 ms
   "2935RS001A01T03.DQ.AL_L2" : Bool AT %DB5079.DBX16.4, 500 ms
   "2935RS001A01T03.DQ.AL_L3" : Bool AT %DB5079.DBX16.5, 500 ms
   "2935RS001A01T03.DQ.SIG_OK" : Bool AT %DB5079.DBX16.6, 500 ms
   "2935RS001A01T03.DQ.LIM_H2" : Bool AT %DB5079.DBX16.7, 500 ms
   "2935RS001A01T03.DQ.LIM_H1" : Bool AT %DB5079.DBX17.0, 500 ms
   "2935RS001A01T03.DQ.LIM_L1" : Bool AT %DB5079.DBX17.1, 500 ms
   "2935RS001A01T03.DQ.LIM_L2" : Bool AT %DB5079.DBX17.2, 500 ms
   "2935RS001A01T03.DQ.GR_P" : Bool AT %DB5079.DBX17.3, 500 ms
   "2935RS001A01T03.DQ.GR_N" : Bool AT %DB5079.DBX17.4, 500 ms
   "2935RS001A01T03.I.IN" : Real AT %DB5079.DBD2, 500 ms
   "2935RS001A01T03.I.SIG_TYPE" : Int AT %DB5079.DBW0, 500 ms
   "2935RS001A01T03.I.FI_BUS" : Byte AT %DB5079.DBB6, 500 ms
   "2935RS001A01T03.DI.U_RANGE" : Bool AT %DB5079.DBX7.0, 500 ms
   "2935RS001A01T03.DI.O_RANGE" : Bool AT %DB5079.DBX7.1, 500 ms
   "2935RS001A01T03.DI.SIG_FAULT" : Bool AT %DB5079.DBX7.2, 500 ms
   "2935RS001A01T03.DI.EnConfig" : Bool AT %DB5079.DBX7.3, 500 ms
   "2935RS001A01T03.DI.AEN" : Bool AT %DB5079.DBX7.4, 500 ms
   "2935RS001A01T03.DI.AL_SUPR" : Bool AT %DB5079.DBX7.5, 500 ms
   "2935RS001A01T03.Q.PV_NORM" : Real AT %DB5079.DBD8, 500 ms
   "2935RS001A01T03.Q.PV_SCAL" : Real AT %DB5079.DBD12, 500 ms
   "2935RS001A01T03.ParentInfo" : TextRef, internal   // Имя родителя для попап окна, вкладка инфо. При експорте из ECS через скрипт заполняется автоматически, если теги копируются в ручную то требуется в ручную задатать свойство Start Value

HMI tags "2935RS001A01T04"
   "2935RS001A01T04.MSW" : 52809b66-421d-457f-8884-6f7a49d4e247 AT %DB5080.DBX18.0, 500 ms
   "2935RS001A01T04.DefaultText" : TextRef, internal   // Заголовок POPUP окна. При експорте из ECS через скрипт заполняется автоматически, если теги копируются в ручную то требуется в ручную задатать свойство Start Value
   "2935RS001A01T04.BlockInfo" : Array [0..2] of Int AT %DB5080.DBX38.0, 500 ms
   "2935RS001A01T04.StatusWork" : Int AT %DB5080.DBW242, 500 ms
   "2935RS001A01T04.FP_PARAM.DampingTime" : Int AT %DB5080.DBW50, 500 ms
   "2935RS001A01T04.FP_PARAM.Force_Value" : Real AT %DB5080.DBD52, 500 ms
   "2935RS001A01T04.FP_PARAM.Scale_Min" : Real AT %DB5080.DBD56, 500 ms
   "2935RS001A01T04.FP_PARAM.Scale_Max" : Real AT %DB5080.DBD60, 500 ms
   "2935RS001A01T04.FP_PARAM.Gradient" : Real AT %DB5080.DBD64, 500 ms
   "2935RS001A01T04.FP_PARAM.Grad_Pos" : Real AT %DB5080.DBD68, 500 ms
   "2935RS001A01T04.FP_PARAM.Grad_Neg" : Real AT %DB5080.DBD72, 500 ms
   "2935RS001A01T04.FP_PARAM.Grad_X" : Real AT %DB5080.DBD76, 500 ms
   "2935RS001A01T04.FP_PARAM.Gradient_Time_Pre" : Int AT %DB5080.DBW80, 500 ms
   "2935RS001A01T04.FP_PARAM.Gradient_Time_ACC" : Int AT %DB5080.DBW82, 500 ms
   "2935RS001A01T04.FP_PARAM.Alarm_Hyst" : Real AT %DB5080.DBD84, 500 ms
   "2935RS001A01T04.FP_PARAM.AlarmLimit_H3" : Real AT %DB5080.DBD88, 500 ms
   "2935RS001A01T04.FP_PARAM.AlarmLimit_H2" : Real AT %DB5080.DBD92, 500 ms
   "2935RS001A01T04.FP_PARAM.AlarmLimit_H1" : Real AT %DB5080.DBD96, 500 ms
   "2935RS001A01T04.FP_PARAM.AlarmLimit_L1" : Real AT %DB5080.DBD100, 500 ms
   "2935RS001A01T04.FP_PARAM.AlarmLimit_L2" : Real AT %DB5080.DBD104, 500 ms
   "2935RS001A01T04.FP_PARAM.AlarmLimit_L3" : Real AT %DB5080.DBD108, 500 ms
   "2935RS001A01T04.FP_PARAM.AlarmDelay_H3_Pre" : Int AT %DB5080.DBW112, 500 ms
   "2935RS001A01T04.FP_PARAM.AlarmDelay_H3_Acc" : Int AT %DB5080.DBW114, 500 ms
   "2935RS001A01T04.FP_PARAM.AlarmDelay_H2_Pre" : Int AT %DB5080.DBW116, 500 ms
   "2935RS001A01T04.FP_PARAM.AlarmDelay_H2_Acc" : Int AT %DB5080.DBW118, 500 ms
   "2935RS001A01T04.FP_PARAM.AlarmDelay_H1_Pre" : Int AT %DB5080.DBW120, 500 ms
   "2935RS001A01T04.FP_PARAM.AlarmDelay_H1_Acc" : Int AT %DB5080.DBW122, 500 ms
   "2935RS001A01T04.FP_PARAM.AlarmDelay_L1_Pre" : Int AT %DB5080.DBW124, 500 ms
   "2935RS001A01T04.FP_PARAM.AlarmDelay_L1_Acc" : Int AT %DB5080.DBW126, 500 ms
   "2935RS001A01T04.FP_PARAM.AlarmDelay_L2_Pre" : Int AT %DB5080.DBW128, 500 ms
   "2935RS001A01T04.FP_PARAM.AlarmDelay_L2_Acc" : Int AT %DB5080.DBW130, 500 ms
   "2935RS001A01T04.FP_PARAM.AlarmDelay_L3_Pre" : Int AT %DB5080.DBW132, 500 ms
   "2935RS001A01T04.FP_PARAM.AlarmDelay_L3_Acc" : Int AT %DB5080.DBW134, 500 ms
   "2935RS001A01T04.FP_PARAM.OpenLoopDelay_Pre" : Int AT %DB5080.DBW136, 500 ms
   "2935RS001A01T04.FP_PARAM.OpenLoopDelay_Acc" : Int AT %DB5080.DBW138, 500 ms
   "2935RS001A01T04.FP_PARAM.OverRangeDelay_Pre" : Int AT %DB5080.DBW140, 500 ms
   "2935RS001A01T04.FP_PARAM.OverRangeDelay_Acc" : Int AT %DB5080.DBW142, 500 ms
   "2935RS001A01T04.FP_PARAM.AuxLimit_H2_Value" : Real AT %DB5080.DBD144, 500 ms
   "2935RS001A01T04.FP_PARAM.AuxLimit_H1_Value" : Real AT %DB5080.DBD148, 500 ms
   "2935RS001A01T04.FP_PARAM.AuxLimit_L2_Value" : Real AT %DB5080.DBD152, 500 ms
   "2935RS001A01T04.FP_PARAM.AuxLimit_L1_Value" : Real AT %DB5080.DBD156, 500 ms
   "2935RS001A01T04.Unit" : TextRef, internal   // Еденицы измерения При експорте из ECS через скрипт заполняется автоматически, если теги копируются в ручную то требуется задатать свойство Text
   "2935RS001A01T04.Decimals" : TextRef, internal   // Формат отображения При експорте из ECS через скрипт, заполняется автоматически. Если теги копируются в ручную то требуется задатать свойство Text s999999.9
   "2935RS001A01T04.FP_EN.Square" : Bool AT %DB5080.DBX46.0, 500 ms
   "2935RS001A01T04.FP_EN.SquareRoot" : Bool AT %DB5080.DBX46.1, 500 ms
   "2935RS001A01T04.FP_EN.ParentSupress" : Bool AT %DB5080.DBX46.2, 500 ms
   "2935RS001A01T04.FP_EN.ParentSupressUnit" : Bool AT %DB5080.DBX46.3, 500 ms
   "2935RS001A01T04.FP_EN.Force" : Bool AT %DB5080.DBX46.4, 500 ms
   "2935RS001A01T04.FP_EN.Damping" : Bool AT %DB5080.DBX46.5, 500 ms
   "2935RS001A01T04.FP_EN.Gradient_Pos" : Bool AT %DB5080.DBX46.6, 500 ms
   "2935RS001A01T04.FP_EN.Gradient_Neg" : Bool AT %DB5080.DBX46.7, 500 ms
   "2935RS001A01T04.FP_EN.Hysteresis" : Bool AT %DB5080.DBX47.0, 500 ms
   "2935RS001A01T04.FP_EN.Alarm_H3" : Bool AT %DB5080.DBX47.1, 500 ms
   "2935RS001A01T04.FP_EN.Alarm_H2" : Bool AT %DB5080.DBX47.2, 500 ms
   "2935RS001A01T04.FP_EN.Alarm_H1" : Bool AT %DB5080.DBX47.3, 500 ms
   "2935RS001A01T04.FP_EN.Alarm_L1" : Bool AT %DB5080.DBX47.4, 500 ms
   "2935RS001A01T04.FP_EN.Alarm_L2" : Bool AT %DB5080.DBX47.5, 500 ms
   "2935RS001A01T04.FP_EN.Alarm_L3" : Bool AT %DB5080.DBX47.6, 500 ms
   "2935RS001A01T04.FP_EN.AlarmDelay_H3" : Bool AT %DB5080.DBX47.7, 500 ms
   "2935RS001A01T04.FP_EN.AlarmDelay_H2" : Bool AT %DB5080.DBX48.0, 500 ms
   "2935RS001A01T04.FP_EN.AlarmDelay_H1" : Bool AT %DB5080.DBX48.1, 500 ms
   "2935RS001A01T04.FP_EN.AlarmDelay_L1" : Bool AT %DB5080.DBX48.2, 500 ms
   "2935RS001A01T04.FP_EN.AlarmDelay_L2" : Bool AT %DB5080.DBX48.3, 500 ms
   "2935RS001A01T04.FP_EN.AlarmDelay_L3" : Bool AT %DB5080.DBX48.4, 500 ms
   "2935RS001A01T04.FP_EN.ROC_Warn" : Bool AT %DB5080.DBX48.5, 500 ms
   "2935RS001A01T04.FP_EN.U_Range_Warn" : Bool AT %DB5080.DBX48.6, 500 ms
   "2935RS001A01T04.FP_EN.O_Range_Warn" : Bool AT %DB5080.DBX48.7, 500 ms
   "2935RS001A01T04.trend_tag_name" : TextRef, internal   // Еденицы измерения При експорте из ECS через скрипт - заполняется автоматически, если теги копируются в ручную то требуется задатать свойство Text - имя тега для тренда
   "2935RS001A01T04.DQ.AL_H3" : Bool AT %DB5080.DBX16.0, 500 ms
   "2935RS001A01T04.DQ.AL_H2" : Bool AT %DB5080.DBX16.1, 500 ms
   "2935RS001A01T04.DQ.AL_H1" : Bool AT %DB5080.DBX16.2, 500 ms
   "2935RS001A01T04.DQ.AL_L1" : Bool AT %DB5080.DBX16.3, 500 ms
   "2935RS001A01T04.DQ.AL_L2" : Bool AT %DB5080.DBX16.4, 500 ms
   "2935RS001A01T04.DQ.AL_L3" : Bool AT %DB5080.DBX16.5, 500 ms
   "2935RS001A01T04.DQ.SIG_OK" : Bool AT %DB5080.DBX16.6, 500 ms
   "2935RS001A01T04.DQ.LIM_H2" : Bool AT %DB5080.DBX16.7, 500 ms
   "2935RS001A01T04.DQ.LIM_H1" : Bool AT %DB5080.DBX17.0, 500 ms
   "2935RS001A01T04.DQ.LIM_L1" : Bool AT %DB5080.DBX17.1, 500 ms
   "2935RS001A01T04.DQ.LIM_L2" : Bool AT %DB5080.DBX17.2, 500 ms
   "2935RS001A01T04.DQ.GR_P" : Bool AT %DB5080.DBX17.3, 500 ms
   "2935RS001A01T04.DQ.GR_N" : Bool AT %DB5080.DBX17.4, 500 ms
   "2935RS001A01T04.I.IN" : Real AT %DB5080.DBD2, 500 ms
   "2935RS001A01T04.I.SIG_TYPE" : Int AT %DB5080.DBW0, 500 ms
   "2935RS001A01T04.I.FI_BUS" : Byte AT %DB5080.DBB6, 500 ms
   "2935RS001A01T04.DI.U_RANGE" : Bool AT %DB5080.DBX7.0, 500 ms
   "2935RS001A01T04.DI.O_RANGE" : Bool AT %DB5080.DBX7.1, 500 ms
   "2935RS001A01T04.DI.SIG_FAULT" : Bool AT %DB5080.DBX7.2, 500 ms
   "2935RS001A01T04.DI.EnConfig" : Bool AT %DB5080.DBX7.3, 500 ms
   "2935RS001A01T04.DI.AEN" : Bool AT %DB5080.DBX7.4, 500 ms
   "2935RS001A01T04.DI.AL_SUPR" : Bool AT %DB5080.DBX7.5, 500 ms
   "2935RS001A01T04.Q.PV_NORM" : Real AT %DB5080.DBD8, 500 ms
   "2935RS001A01T04.Q.PV_SCAL" : Real AT %DB5080.DBD12, 500 ms
   "2935RS001A01T04.ParentInfo" : TextRef, internal   // Имя родителя для попап окна, вкладка инфо. При експорте из ECS через скрипт заполняется автоматически, если теги копируются в ручную то требуется в ручную задатать свойство Start Value

